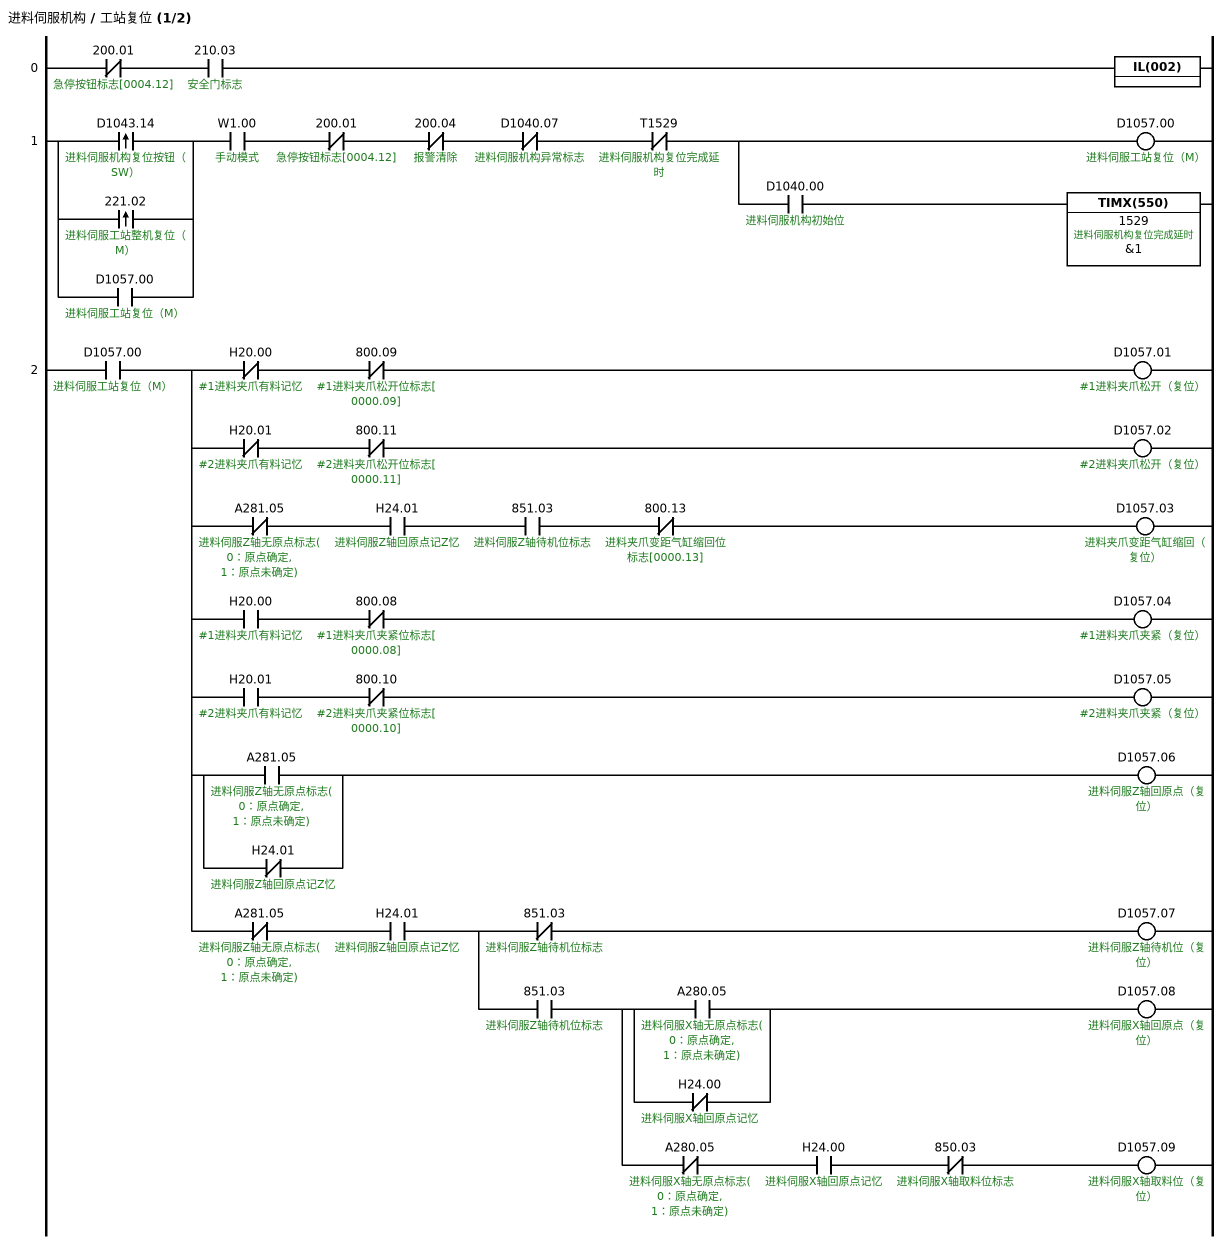
; rung 0
LDNOT 200.01  ; 急停按钮标志[0004.12]
AND 210.03  ; 安全门标志
IL(002)
; rung 1
@LD D1043.14  ; 进料伺服机构复位按钮（SW）
@OR 221.02  ; 进料伺服工站整机复位（M）
OR D1057.00  ; 进料伺服工站复位（M）
AND W1.00  ; 手动模式
ANDNOT 200.01  ; 急停按钮标志[0004.12]
ANDNOT 200.04  ; 报警清除
ANDNOT D1040.07  ; 进料伺服机构异常标志
ANDNOT T1529  ; 进料伺服机构复位完成延时
OUT D1057.00  ; 进料伺服工站复位（M）
AND D1040.00  ; 进料伺服机构初始位
TIMX(550) 1529 &1  ; 进料伺服机构复位完成延时
; rung 2
LD D1057.00  ; 进料伺服工站复位（M）
OUT TR0
ANDNOT H20.00  ; #1进料夹爪有料记忆
ANDNOT 800.09  ; #1进料夹爪松开位标志[0000.09]
OUT D1057.01  ; #1进料夹爪松开（复位）
LD TR0
ANDNOT H20.01  ; #2进料夹爪有料记忆
ANDNOT 800.11  ; #2进料夹爪松开位标志[0000.11]
OUT D1057.02  ; #2进料夹爪松开（复位）
LD TR0
ANDNOT A281.05  ; 进料伺服Z轴无原点标志(0：原点确定,1：原点未确定)
AND H24.01  ; 进料伺服Z轴回原点记Z忆
AND 851.03  ; 进料伺服Z轴待机位标志
ANDNOT 800.13  ; 进料夹爪变距气缸缩回位标志[0000.13]
OUT D1057.03  ; 进料夹爪变距气缸缩回（复位）
LD TR0
AND H20.00  ; #1进料夹爪有料记忆
ANDNOT 800.08  ; #1进料夹爪夹紧位标志[0000.08]
OUT D1057.04  ; #1进料夹爪夹紧（复位）
LD TR0
AND H20.01  ; #2进料夹爪有料记忆
ANDNOT 800.10  ; #2进料夹爪夹紧位标志[0000.10]
OUT D1057.05  ; #2进料夹爪夹紧（复位）
LD TR0
LD A281.05  ; 进料伺服Z轴无原点标志(0：原点确定,1：原点未确定)
ORNOT H24.01  ; 进料伺服Z轴回原点记Z忆
ANDLD
OUT D1057.06  ; 进料伺服Z轴回原点（复位）
LD TR0
ANDNOT A281.05  ; 进料伺服Z轴无原点标志(0：原点确定,1：原点未确定)
AND H24.01  ; 进料伺服Z轴回原点记Z忆
OUT TR0
ANDNOT 851.03  ; 进料伺服Z轴待机位标志
OUT D1057.07  ; 进料伺服Z轴待机位（复位）
LD TR0
AND 851.03  ; 进料伺服Z轴待机位标志
OUT TR0
LD A280.05  ; 进料伺服X轴无原点标志(0：原点确定,1：原点未确定)
ORNOT H24.00  ; 进料伺服X轴回原点记忆
ANDLD
OUT D1057.08  ; 进料伺服X轴回原点（复位）
LD TR0
ANDNOT A280.05  ; 进料伺服X轴无原点标志(0：原点确定,1：原点未确定)
AND H24.00  ; 进料伺服X轴回原点记忆
ANDNOT 850.03  ; 进料伺服X轴取料位标志
OUT D1057.09  ; 进料伺服X轴取料位（复位）

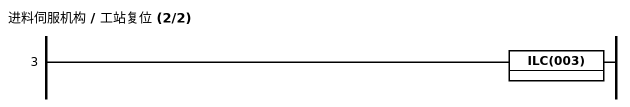
; rung 3
ILC(003)

### Section 指示灯

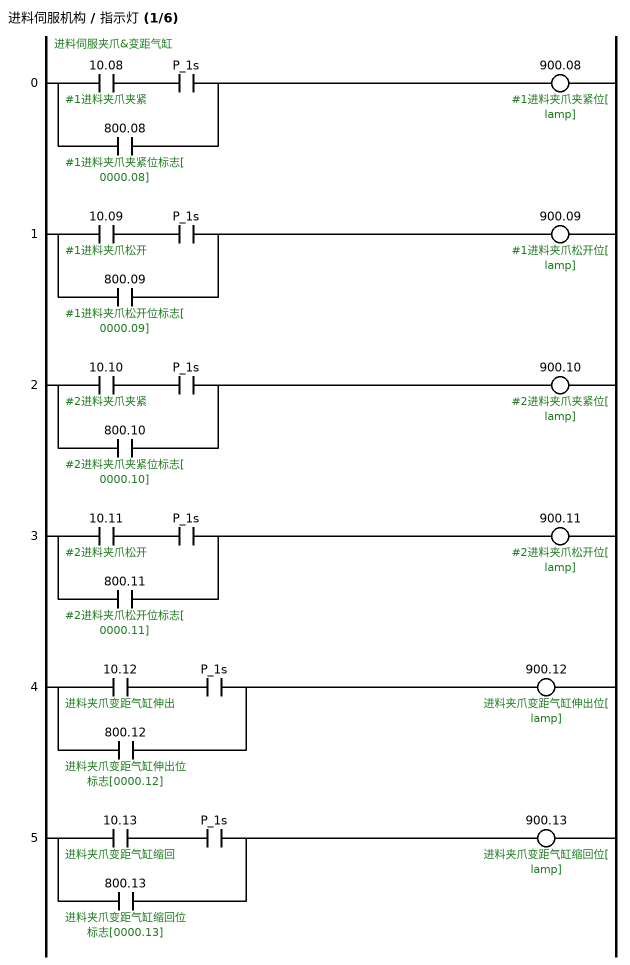
; rung 0: 进料伺服夹爪&变距气缸
LD 10.08  ; #1进料夹爪夹紧
AND P_1s
OR 800.08  ; #1进料夹爪夹紧位标志[0000.08]
OUT 900.08  ; #1进料夹爪夹紧位[lamp]
; rung 1
LD 10.09  ; #1进料夹爪松开
AND P_1s
OR 800.09  ; #1进料夹爪松开位标志[0000.09]
OUT 900.09  ; #1进料夹爪松开位[lamp]
; rung 2
LD 10.10  ; #2进料夹爪夹紧
AND P_1s
OR 800.10  ; #2进料夹爪夹紧位标志[0000.10]
OUT 900.10  ; #2进料夹爪夹紧位[lamp]
; rung 3
LD 10.11  ; #2进料夹爪松开
AND P_1s
OR 800.11  ; #2进料夹爪松开位标志[0000.11]
OUT 900.11  ; #2进料夹爪松开位[lamp]
; rung 4
LD 10.12  ; 进料夹爪变距气缸伸出
AND P_1s
OR 800.12  ; 进料夹爪变距气缸伸出位标志[0000.12]
OUT 900.12  ; 进料夹爪变距气缸伸出位[lamp]
; rung 5
LD 10.13  ; 进料夹爪变距气缸缩回
AND P_1s
OR 800.13  ; 进料夹爪变距气缸缩回位标志[0000.13]
OUT 900.13  ; 进料夹爪变距气缸缩回位[lamp]

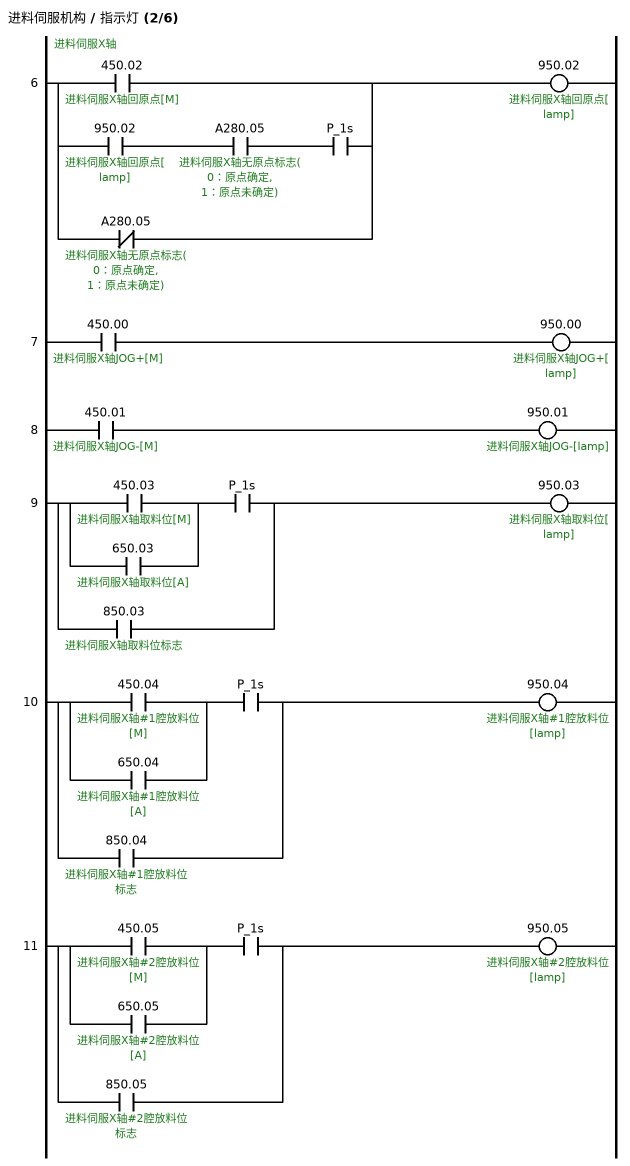
; rung 6: 进料伺服X轴
LD 450.02  ; 进料伺服X轴回原点[M]
LD 950.02  ; 进料伺服X轴回原点[lamp]
AND A280.05  ; 进料伺服X轴无原点标志(0：原点确定,1：原点未确定)
AND P_1s
ORLD
ORNOT A280.05  ; 进料伺服X轴无原点标志(0：原点确定,1：原点未确定)
OUT 950.02  ; 进料伺服X轴回原点[lamp]
; rung 7
LD 450.00  ; 进料伺服X轴JOG+[M]
OUT 950.00  ; 进料伺服X轴JOG+[lamp]
; rung 8
LD 450.01  ; 进料伺服X轴JOG-[M]
OUT 950.01  ; 进料伺服X轴JOG-[lamp]
; rung 9
LD 450.03  ; 进料伺服X轴取料位[M]
OR 650.03  ; 进料伺服X轴取料位[A]
AND P_1s
OR 850.03  ; 进料伺服X轴取料位标志
OUT 950.03  ; 进料伺服X轴取料位[lamp]
; rung 10
LD 450.04  ; 进料伺服X轴#1腔放料位[M]
OR 650.04  ; 进料伺服X轴#1腔放料位[A]
AND P_1s
OR 850.04  ; 进料伺服X轴#1腔放料位标志
OUT 950.04  ; 进料伺服X轴#1腔放料位[lamp]
; rung 11
LD 450.05  ; 进料伺服X轴#2腔放料位[M]
OR 650.05  ; 进料伺服X轴#2腔放料位[A]
AND P_1s
OR 850.05  ; 进料伺服X轴#2腔放料位标志
OUT 950.05  ; 进料伺服X轴#2腔放料位[lamp]

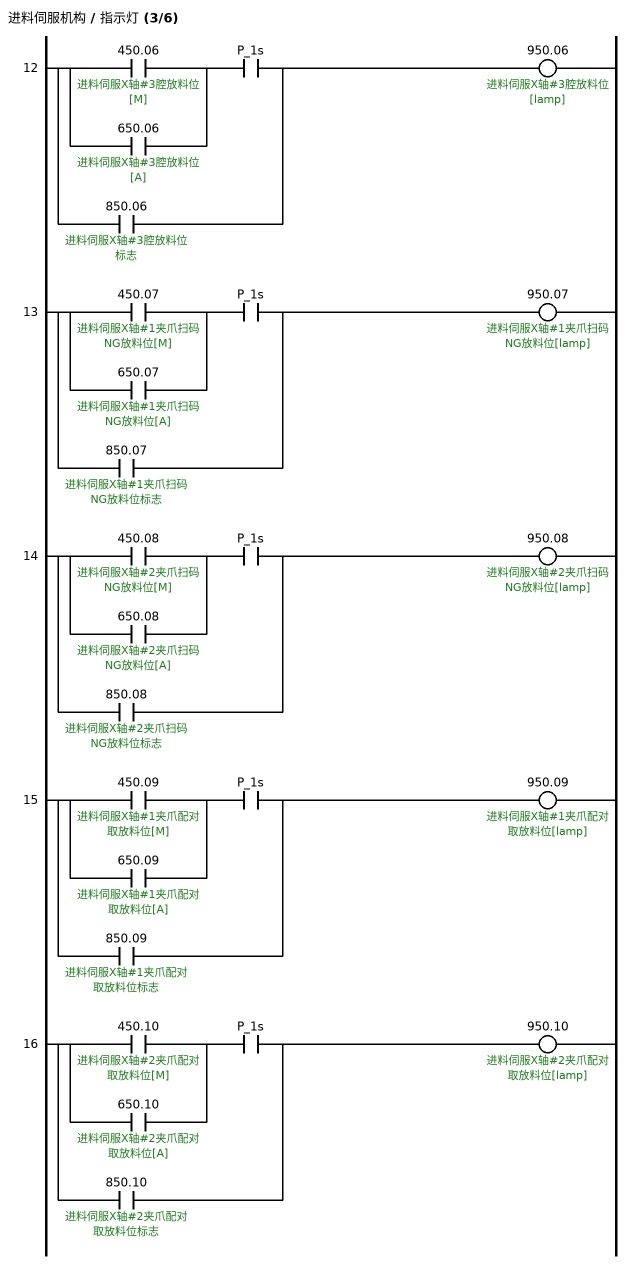
; rung 12
LD 450.06  ; 进料伺服X轴#3腔放料位[M]
OR 650.06  ; 进料伺服X轴#3腔放料位[A]
AND P_1s
OR 850.06  ; 进料伺服X轴#3腔放料位标志
OUT 950.06  ; 进料伺服X轴#3腔放料位[lamp]
; rung 13
LD 450.07  ; 进料伺服X轴#1夹爪扫码NG放料位[M]
OR 650.07  ; 进料伺服X轴#1夹爪扫码NG放料位[A]
AND P_1s
OR 850.07  ; 进料伺服X轴#1夹爪扫码NG放料位标志
OUT 950.07  ; 进料伺服X轴#1夹爪扫码NG放料位[lamp]
; rung 14
LD 450.08  ; 进料伺服X轴#2夹爪扫码NG放料位[M]
OR 650.08  ; 进料伺服X轴#2夹爪扫码NG放料位[A]
AND P_1s
OR 850.08  ; 进料伺服X轴#2夹爪扫码NG放料位标志
OUT 950.08  ; 进料伺服X轴#2夹爪扫码NG放料位[lamp]
; rung 15
LD 450.09  ; 进料伺服X轴#1夹爪配对取放料位[M]
OR 650.09  ; 进料伺服X轴#1夹爪配对取放料位[A]
AND P_1s
OR 850.09  ; 进料伺服X轴#1夹爪配对取放料位标志
OUT 950.09  ; 进料伺服X轴#1夹爪配对取放料位[lamp]
; rung 16
LD 450.10  ; 进料伺服X轴#2夹爪配对取放料位[M]
OR 650.10  ; 进料伺服X轴#2夹爪配对取放料位[A]
AND P_1s
OR 850.10  ; 进料伺服X轴#2夹爪配对取放料位标志
OUT 950.10  ; 进料伺服X轴#2夹爪配对取放料位[lamp]

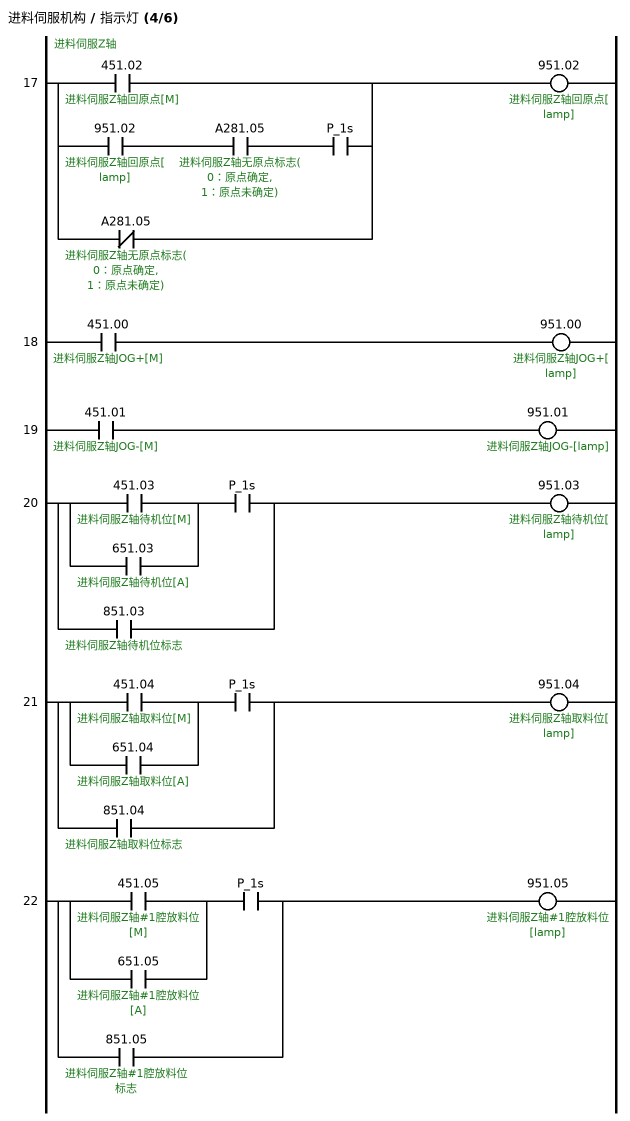
; rung 17: 进料伺服Z轴
LD 451.02  ; 进料伺服Z轴回原点[M]
LD 951.02  ; 进料伺服Z轴回原点[lamp]
AND A281.05  ; 进料伺服Z轴无原点标志(0：原点确定,1：原点未确定)
AND P_1s
ORLD
ORNOT A281.05  ; 进料伺服Z轴无原点标志(0：原点确定,1：原点未确定)
OUT 951.02  ; 进料伺服Z轴回原点[lamp]
; rung 18
LD 451.00  ; 进料伺服Z轴JOG+[M]
OUT 951.00  ; 进料伺服Z轴JOG+[lamp]
; rung 19
LD 451.01  ; 进料伺服Z轴JOG-[M]
OUT 951.01  ; 进料伺服Z轴JOG-[lamp]
; rung 20
LD 451.03  ; 进料伺服Z轴待机位[M]
OR 651.03  ; 进料伺服Z轴待机位[A]
AND P_1s
OR 851.03  ; 进料伺服Z轴待机位标志
OUT 951.03  ; 进料伺服Z轴待机位[lamp]
; rung 21
LD 451.04  ; 进料伺服Z轴取料位[M]
OR 651.04  ; 进料伺服Z轴取料位[A]
AND P_1s
OR 851.04  ; 进料伺服Z轴取料位标志
OUT 951.04  ; 进料伺服Z轴取料位[lamp]
; rung 22
LD 451.05  ; 进料伺服Z轴#1腔放料位[M]
OR 651.05  ; 进料伺服Z轴#1腔放料位[A]
AND P_1s
OR 851.05  ; 进料伺服Z轴#1腔放料位标志
OUT 951.05  ; 进料伺服Z轴#1腔放料位[lamp]

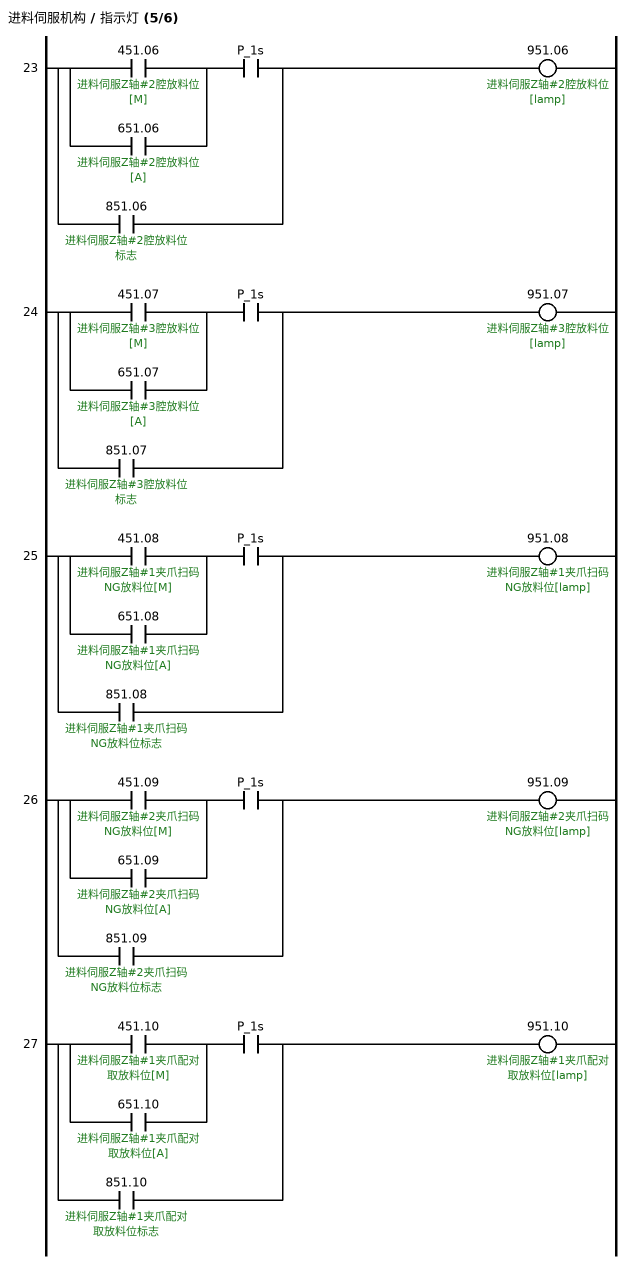
; rung 23
LD 451.06  ; 进料伺服Z轴#2腔放料位[M]
OR 651.06  ; 进料伺服Z轴#2腔放料位[A]
AND P_1s
OR 851.06  ; 进料伺服Z轴#2腔放料位标志
OUT 951.06  ; 进料伺服Z轴#2腔放料位[lamp]
; rung 24
LD 451.07  ; 进料伺服Z轴#3腔放料位[M]
OR 651.07  ; 进料伺服Z轴#3腔放料位[A]
AND P_1s
OR 851.07  ; 进料伺服Z轴#3腔放料位标志
OUT 951.07  ; 进料伺服Z轴#3腔放料位[lamp]
; rung 25
LD 451.08  ; 进料伺服Z轴#1夹爪扫码NG放料位[M]
OR 651.08  ; 进料伺服Z轴#1夹爪扫码NG放料位[A]
AND P_1s
OR 851.08  ; 进料伺服Z轴#1夹爪扫码NG放料位标志
OUT 951.08  ; 进料伺服Z轴#1夹爪扫码NG放料位[lamp]
; rung 26
LD 451.09  ; 进料伺服Z轴#2夹爪扫码NG放料位[M]
OR 651.09  ; 进料伺服Z轴#2夹爪扫码NG放料位[A]
AND P_1s
OR 851.09  ; 进料伺服Z轴#2夹爪扫码NG放料位标志
OUT 951.09  ; 进料伺服Z轴#2夹爪扫码NG放料位[lamp]
; rung 27
LD 451.10  ; 进料伺服Z轴#1夹爪配对取放料位[M]
OR 651.10  ; 进料伺服Z轴#1夹爪配对取放料位[A]
AND P_1s
OR 851.10  ; 进料伺服Z轴#1夹爪配对取放料位标志
OUT 951.10  ; 进料伺服Z轴#1夹爪配对取放料位[lamp]

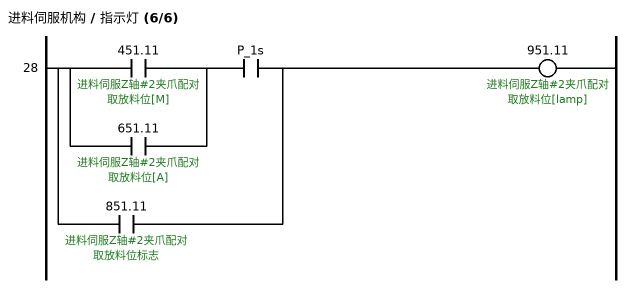
; rung 28
LD 451.11  ; 进料伺服Z轴#2夹爪配对取放料位[M]
OR 651.11  ; 进料伺服Z轴#2夹爪配对取放料位[A]
AND P_1s
OR 851.11  ; 进料伺服Z轴#2夹爪配对取放料位标志
OUT 951.11  ; 进料伺服Z轴#2夹爪配对取放料位[lamp]

### Section 外部输出

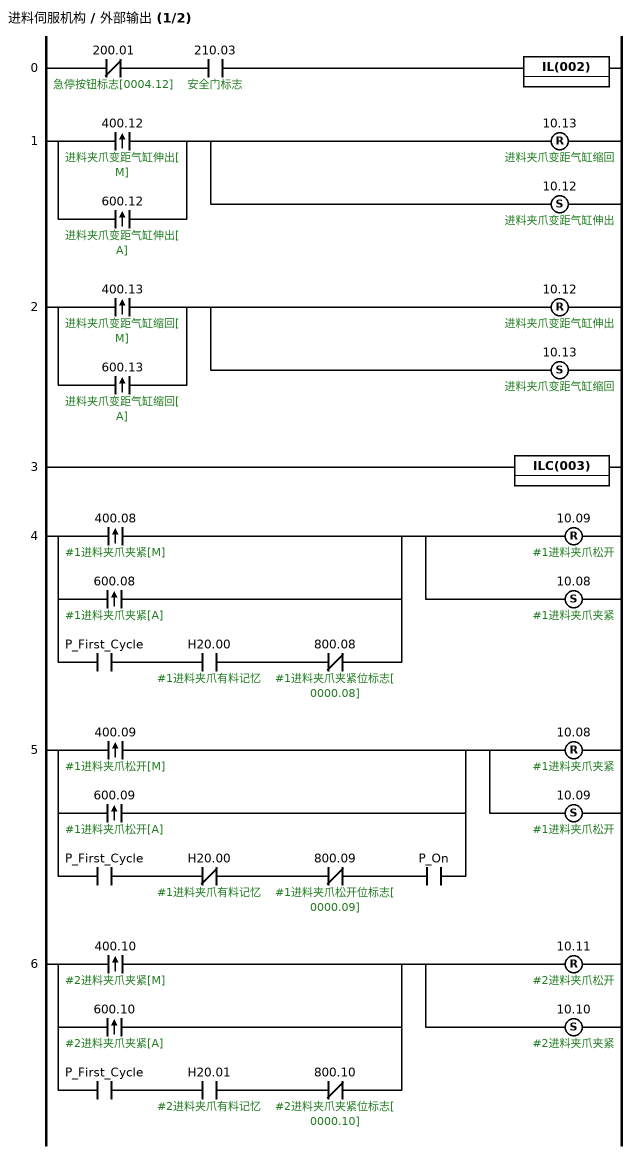
; rung 0
LDNOT 200.01  ; 急停按钮标志[0004.12]
AND 210.03  ; 安全门标志
IL(002)
; rung 1
@LD 400.12  ; 进料夹爪变距气缸伸出[M]
@OR 600.12  ; 进料夹爪变距气缸伸出[A]
RSET 10.13  ; 进料夹爪变距气缸缩回
SET 10.12  ; 进料夹爪变距气缸伸出
; rung 2
@LD 400.13  ; 进料夹爪变距气缸缩回[M]
@OR 600.13  ; 进料夹爪变距气缸缩回[A]
RSET 10.12  ; 进料夹爪变距气缸伸出
SET 10.13  ; 进料夹爪变距气缸缩回
; rung 3
ILC(003)
; rung 4
@LD 400.08  ; #1进料夹爪夹紧[M]
@OR 600.08  ; #1进料夹爪夹紧[A]
LD P_First_Cycle
AND H20.00  ; #1进料夹爪有料记忆
ANDNOT 800.08  ; #1进料夹爪夹紧位标志[0000.08]
ORLD
RSET 10.09  ; #1进料夹爪松开
SET 10.08  ; #1进料夹爪夹紧
; rung 5
@LD 400.09  ; #1进料夹爪松开[M]
@OR 600.09  ; #1进料夹爪松开[A]
LD P_First_Cycle
ANDNOT H20.00  ; #1进料夹爪有料记忆
ANDNOT 800.09  ; #1进料夹爪松开位标志[0000.09]
AND P_On
ORLD
RSET 10.08  ; #1进料夹爪夹紧
SET 10.09  ; #1进料夹爪松开
; rung 6
@LD 400.10  ; #2进料夹爪夹紧[M]
@OR 600.10  ; #2进料夹爪夹紧[A]
LD P_First_Cycle
AND H20.01  ; #2进料夹爪有料记忆
ANDNOT 800.10  ; #2进料夹爪夹紧位标志[0000.10]
ORLD
RSET 10.11  ; #2进料夹爪松开
SET 10.10  ; #2进料夹爪夹紧

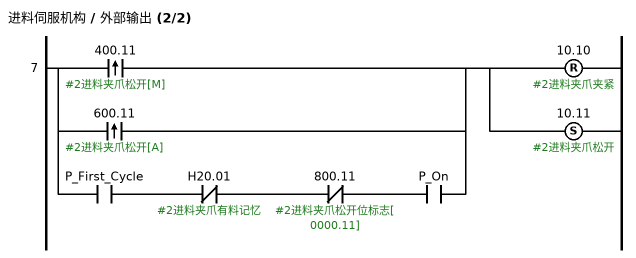
; rung 7
@LD 400.11  ; #2进料夹爪松开[M]
@OR 600.11  ; #2进料夹爪松开[A]
LD P_First_Cycle
ANDNOT H20.01  ; #2进料夹爪有料记忆
ANDNOT 800.11  ; #2进料夹爪松开位标志[0000.11]
AND P_On
ORLD
RSET 10.10  ; #2进料夹爪夹紧
SET 10.11  ; #2进料夹爪松开

### Section END
; rung 0
END(001)

## Program 氦检机构 (cyclic task 3)
Local symbols
UP BOOL

### Section Main

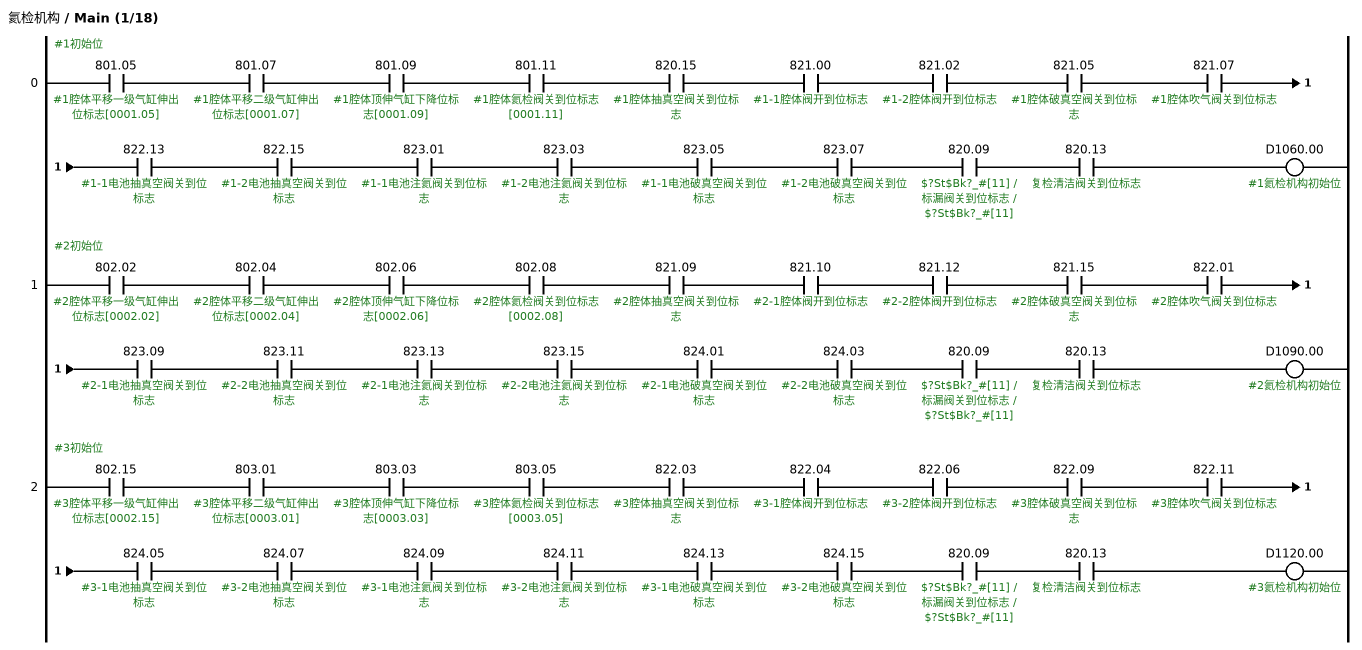
; rung 0: #1初始位
LD 801.05  ; #1腔体平移一级气缸伸出位标志[0001.05]
AND 801.07  ; #1腔体平移二级气缸伸出位标志[0001.07]
AND 801.09  ; #1腔体顶伸气缸下降位标志[0001.09]
AND 801.11  ; #1腔体氦检阀关到位标志[0001.11]
AND 820.15  ; #1腔体抽真空阀关到位标志
AND 821.00  ; #1-1腔体阀开到位标志
AND 821.02  ; #1-2腔体阀开到位标志
AND 821.05  ; #1腔体破真空阀关到位标志
AND 821.07  ; #1腔体吹气阀关到位标志
AND 822.13  ; #1-1电池抽真空阀关到位标志
AND 822.15  ; #1-2电池抽真空阀关到位标志
AND 823.01  ; #1-1电池注氦阀关到位标志
AND 823.03  ; #1-2电池注氦阀关到位标志
AND 823.05  ; #1-1电池破真空阀关到位标志
AND 823.07  ; #1-2电池破真空阀关到位标志
AND 820.09  ; $?St$Bk?_#[11] / 标漏阀关到位标志 / $?St$Bk?_#[11]
AND 820.13  ; 复检清洁阀关到位标志
OUT D1060.00  ; #1氦检机构初始位
; rung 1: #2初始位
LD 802.02  ; #2腔体平移一级气缸伸出位标志[0002.02]
AND 802.04  ; #2腔体平移二级气缸伸出位标志[0002.04]
AND 802.06  ; #2腔体顶伸气缸下降位标志[0002.06]
AND 802.08  ; #2腔体氦检阀关到位标志[0002.08]
AND 821.09  ; #2腔体抽真空阀关到位标志
AND 821.10  ; #2-1腔体阀开到位标志
AND 821.12  ; #2-2腔体阀开到位标志
AND 821.15  ; #2腔体破真空阀关到位标志
AND 822.01  ; #2腔体吹气阀关到位标志
AND 823.09  ; #2-1电池抽真空阀关到位标志
AND 823.11  ; #2-2电池抽真空阀关到位标志
AND 823.13  ; #2-1电池注氦阀关到位标志
AND 823.15  ; #2-2电池注氦阀关到位标志
AND 824.01  ; #2-1电池破真空阀关到位标志
AND 824.03  ; #2-2电池破真空阀关到位标志
AND 820.09  ; $?St$Bk?_#[11] / 标漏阀关到位标志 / $?St$Bk?_#[11]
AND 820.13  ; 复检清洁阀关到位标志
OUT D1090.00  ; #2氦检机构初始位
; rung 2: #3初始位
LD 802.15  ; #3腔体平移一级气缸伸出位标志[0002.15]
AND 803.01  ; #3腔体平移二级气缸伸出位标志[0003.01]
AND 803.03  ; #3腔体顶伸气缸下降位标志[0003.03]
AND 803.05  ; #3腔体氦检阀关到位标志[0003.05]
AND 822.03  ; #3腔体抽真空阀关到位标志
AND 822.04  ; #3-1腔体阀开到位标志
AND 822.06  ; #3-2腔体阀开到位标志
AND 822.09  ; #3腔体破真空阀关到位标志
AND 822.11  ; #3腔体吹气阀关到位标志
AND 824.05  ; #3-1电池抽真空阀关到位标志
AND 824.07  ; #3-2电池抽真空阀关到位标志
AND 824.09  ; #3-1电池注氦阀关到位标志
AND 824.11  ; #3-2电池注氦阀关到位标志
AND 824.13  ; #3-1电池破真空阀关到位标志
AND 824.15  ; #3-2电池破真空阀关到位标志
AND 820.09  ; $?St$Bk?_#[11] / 标漏阀关到位标志 / $?St$Bk?_#[11]
AND 820.13  ; 复检清洁阀关到位标志
OUT D1120.00  ; #3氦检机构初始位

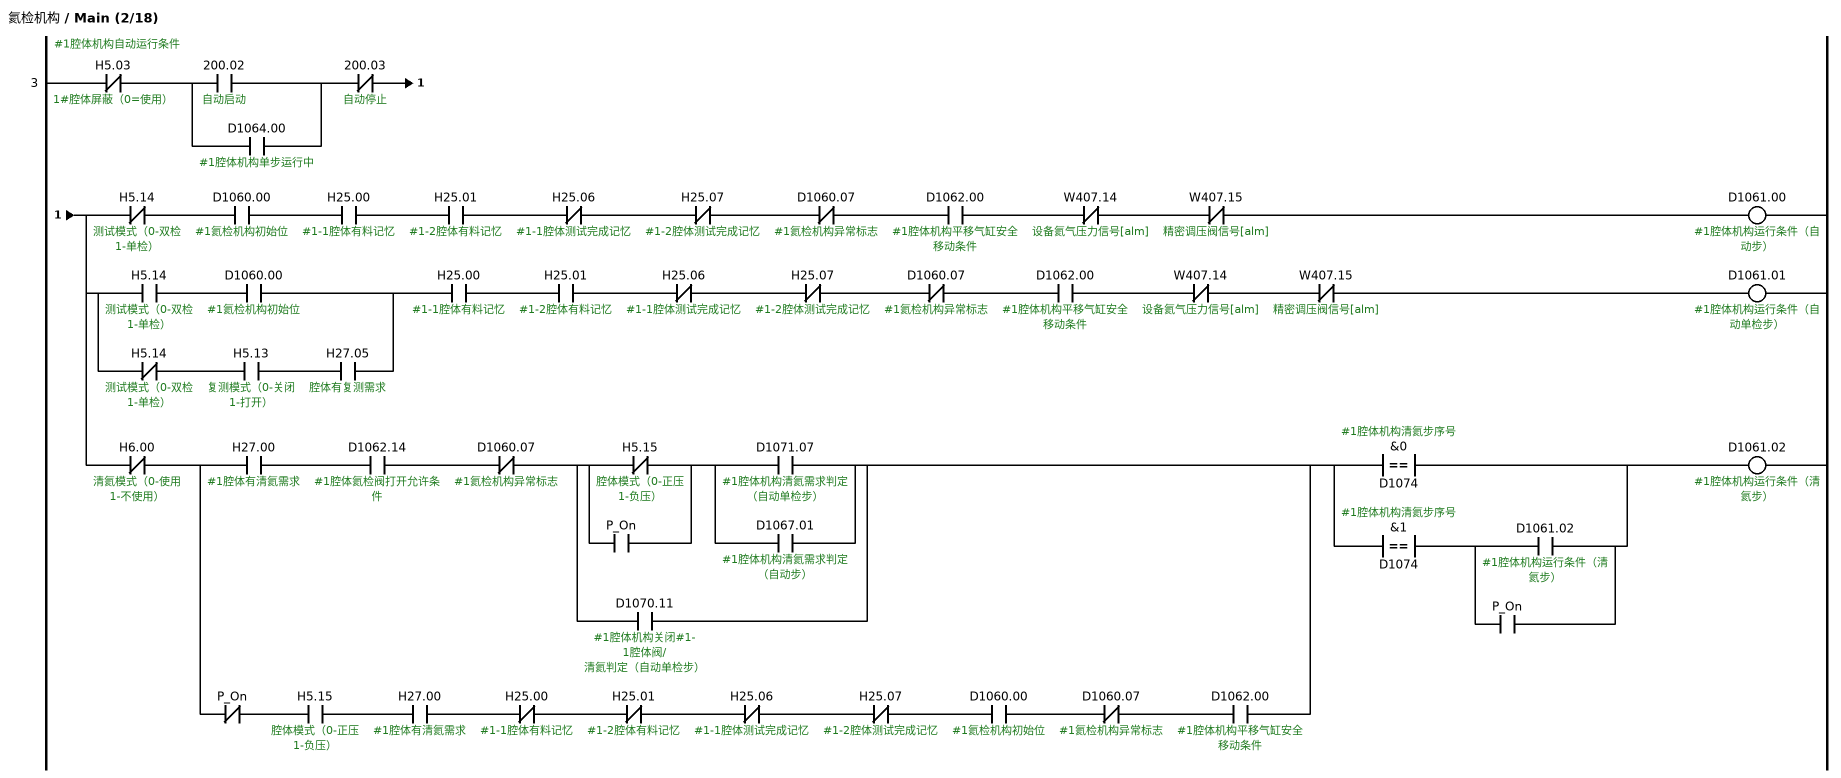
; rung 3: #1腔体机构自动运行条件
LDNOT H5.03  ; 1#腔体屏蔽（0=使用）
LD 200.02  ; 自动启动
OR D1064.00  ; #1腔体机构单步运行中
ANDLD
ANDNOT 200.03  ; 自动停止
OUT TR0
ANDNOT H5.14  ; 测试模式（0-双检 1-单检）
AND D1060.00  ; #1氦检机构初始位
AND H25.00  ; #1-1腔体有料记忆
AND H25.01  ; #1-2腔体有料记忆
ANDNOT H25.06  ; #1-1腔体测试完成记忆
ANDNOT H25.07  ; #1-2腔体测试完成记忆
ANDNOT D1060.07  ; #1氦检机构异常标志
AND D1062.00  ; #1腔体机构平移气缸安全移动条件
ANDNOT W407.14  ; 设备氦气压力信号[alm]
ANDNOT W407.15  ; 精密调压阀信号[alm]
OUT D1061.00  ; #1腔体机构运行条件（自动步）
LD TR0
LD H5.14  ; 测试模式（0-双检 1-单检）
AND D1060.00  ; #1氦检机构初始位
LDNOT H5.14  ; 测试模式（0-双检 1-单检）
AND H5.13  ; 复测模式（0-关闭 1-打开）
AND H27.05  ; 腔体有复测需求
ORLD
ANDLD
AND H25.00  ; #1-1腔体有料记忆
AND H25.01  ; #1-2腔体有料记忆
ANDNOT H25.06  ; #1-1腔体测试完成记忆
ANDNOT H25.07  ; #1-2腔体测试完成记忆
ANDNOT D1060.07  ; #1氦检机构异常标志
AND D1062.00  ; #1腔体机构平移气缸安全移动条件
ANDNOT W407.14  ; 设备氦气压力信号[alm]
ANDNOT W407.15  ; 精密调压阀信号[alm]
OUT D1061.01  ; #1腔体机构运行条件（自动单检步）
LD TR0
ANDNOT H6.00  ; 清氦模式（0-使用 1-不使用）
LD H27.00  ; #1腔体有清氦需求
AND D1062.14  ; #1腔体氦检阀打开允许条件
ANDNOT D1060.07  ; #1氦检机构异常标志
LDNOT H5.15  ; 腔体模式（0-正压 1-负压）
OR P_On
LD D1071.07  ; #1腔体机构清氦需求判定（自动单检步）
OR D1067.01  ; #1腔体机构清氦需求判定（自动步）
ANDLD
OR D1070.11  ; #1腔体机构关闭#1-1腔体阀/清氦判定（自动单检步）
ANDLD
LDNOT P_On
AND H5.15  ; 腔体模式（0-正压 1-负压）
AND H27.00  ; #1腔体有清氦需求
ANDNOT H25.00  ; #1-1腔体有料记忆
ANDNOT H25.01  ; #1-2腔体有料记忆
ANDNOT H25.06  ; #1-1腔体测试完成记忆
ANDNOT H25.07  ; #1-2腔体测试完成记忆
AND D1060.00  ; #1氦检机构初始位
ANDNOT D1060.07  ; #1氦检机构异常标志
AND D1062.00  ; #1腔体机构平移气缸安全移动条件
ORLD
ANDLD
LD=L(301) &0 D1074  ; #1腔体机构清氦步序号
LD=L(301) &1 D1074  ; #1腔体机构清氦步序号
LD D1061.02  ; #1腔体机构运行条件（清氦步）
OR P_On
ANDLD
ORLD
ANDLD
OUT D1061.02  ; #1腔体机构运行条件（清氦步）

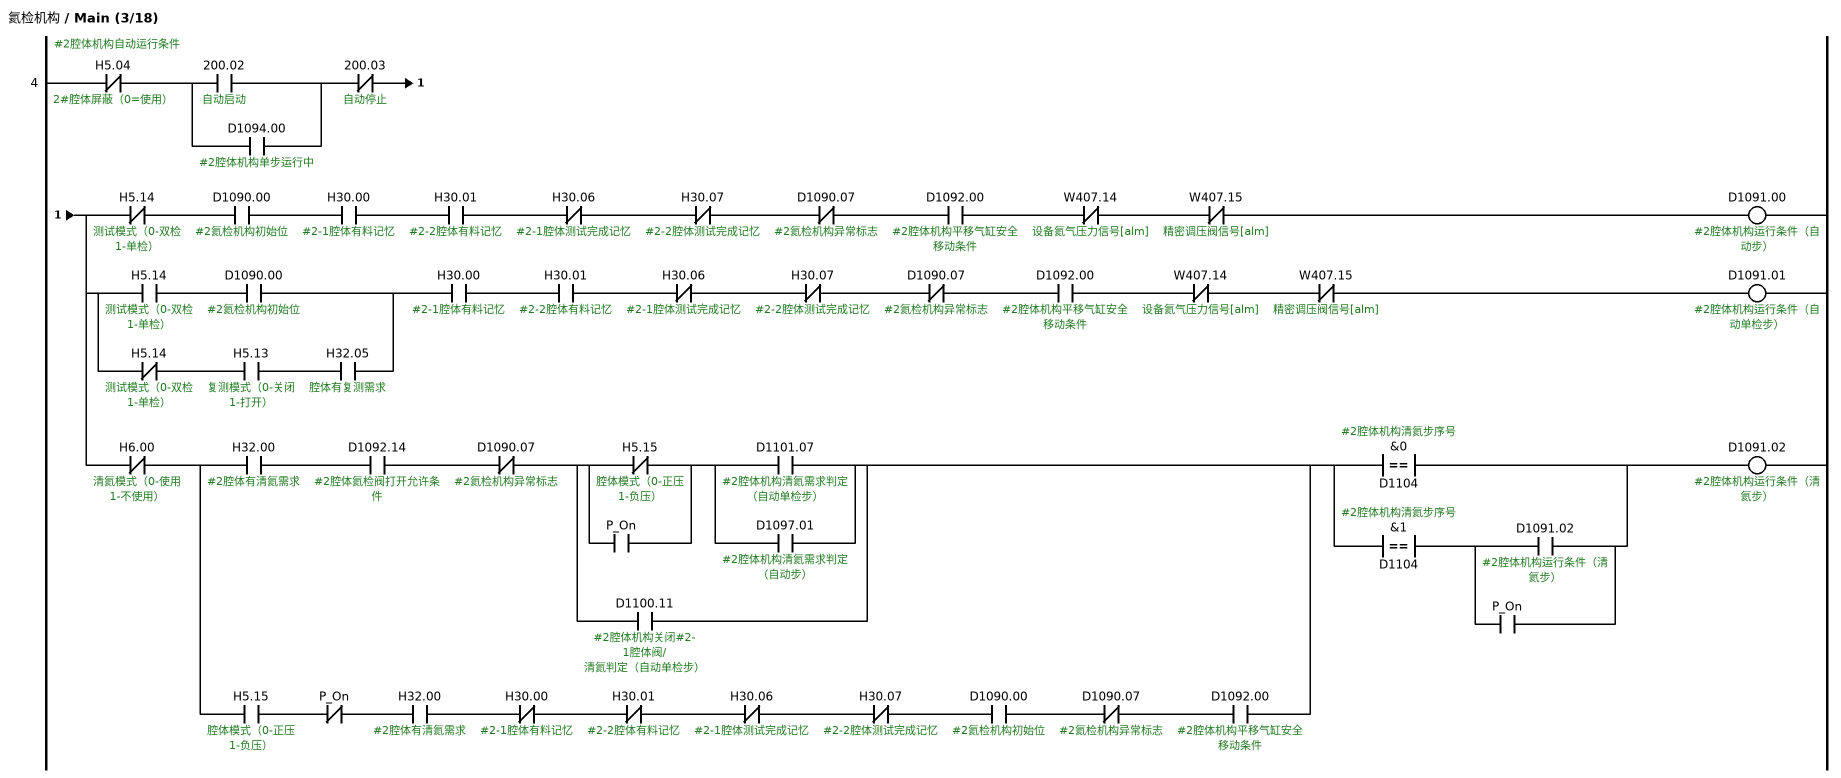
; rung 4: #2腔体机构自动运行条件
LDNOT H5.04  ; 2#腔体屏蔽（0=使用）
LD 200.02  ; 自动启动
OR D1094.00  ; #2腔体机构单步运行中
ANDLD
ANDNOT 200.03  ; 自动停止
OUT TR0
ANDNOT H5.14  ; 测试模式（0-双检 1-单检）
AND D1090.00  ; #2氦检机构初始位
AND H30.00  ; #2-1腔体有料记忆
AND H30.01  ; #2-2腔体有料记忆
ANDNOT H30.06  ; #2-1腔体测试完成记忆
ANDNOT H30.07  ; #2-2腔体测试完成记忆
ANDNOT D1090.07  ; #2氦检机构异常标志
AND D1092.00  ; #2腔体机构平移气缸安全移动条件
ANDNOT W407.14  ; 设备氦气压力信号[alm]
ANDNOT W407.15  ; 精密调压阀信号[alm]
OUT D1091.00  ; #2腔体机构运行条件（自动步）
LD TR0
LD H5.14  ; 测试模式（0-双检 1-单检）
AND D1090.00  ; #2氦检机构初始位
LDNOT H5.14  ; 测试模式（0-双检 1-单检）
AND H5.13  ; 复测模式（0-关闭 1-打开）
AND H32.05  ; 腔体有复测需求
ORLD
ANDLD
AND H30.00  ; #2-1腔体有料记忆
AND H30.01  ; #2-2腔体有料记忆
ANDNOT H30.06  ; #2-1腔体测试完成记忆
ANDNOT H30.07  ; #2-2腔体测试完成记忆
ANDNOT D1090.07  ; #2氦检机构异常标志
AND D1092.00  ; #2腔体机构平移气缸安全移动条件
ANDNOT W407.14  ; 设备氦气压力信号[alm]
ANDNOT W407.15  ; 精密调压阀信号[alm]
OUT D1091.01  ; #2腔体机构运行条件（自动单检步）
LD TR0
ANDNOT H6.00  ; 清氦模式（0-使用 1-不使用）
LD H32.00  ; #2腔体有清氦需求
AND D1092.14  ; #2腔体氦检阀打开允许条件
ANDNOT D1090.07  ; #2氦检机构异常标志
LDNOT H5.15  ; 腔体模式（0-正压 1-负压）
OR P_On
LD D1101.07  ; #2腔体机构清氦需求判定（自动单检步）
OR D1097.01  ; #2腔体机构清氦需求判定（自动步）
ANDLD
OR D1100.11  ; #2腔体机构关闭#2-1腔体阀/清氦判定（自动单检步）
ANDLD
LD H5.15  ; 腔体模式（0-正压 1-负压）
ANDNOT P_On
AND H32.00  ; #2腔体有清氦需求
ANDNOT H30.00  ; #2-1腔体有料记忆
ANDNOT H30.01  ; #2-2腔体有料记忆
ANDNOT H30.06  ; #2-1腔体测试完成记忆
ANDNOT H30.07  ; #2-2腔体测试完成记忆
AND D1090.00  ; #2氦检机构初始位
ANDNOT D1090.07  ; #2氦检机构异常标志
AND D1092.00  ; #2腔体机构平移气缸安全移动条件
ORLD
ANDLD
LD=L(301) &0 D1104  ; #2腔体机构清氦步序号
LD=L(301) &1 D1104  ; #2腔体机构清氦步序号
LD D1091.02  ; #2腔体机构运行条件（清氦步）
OR P_On
ANDLD
ORLD
ANDLD
OUT D1091.02  ; #2腔体机构运行条件（清氦步）

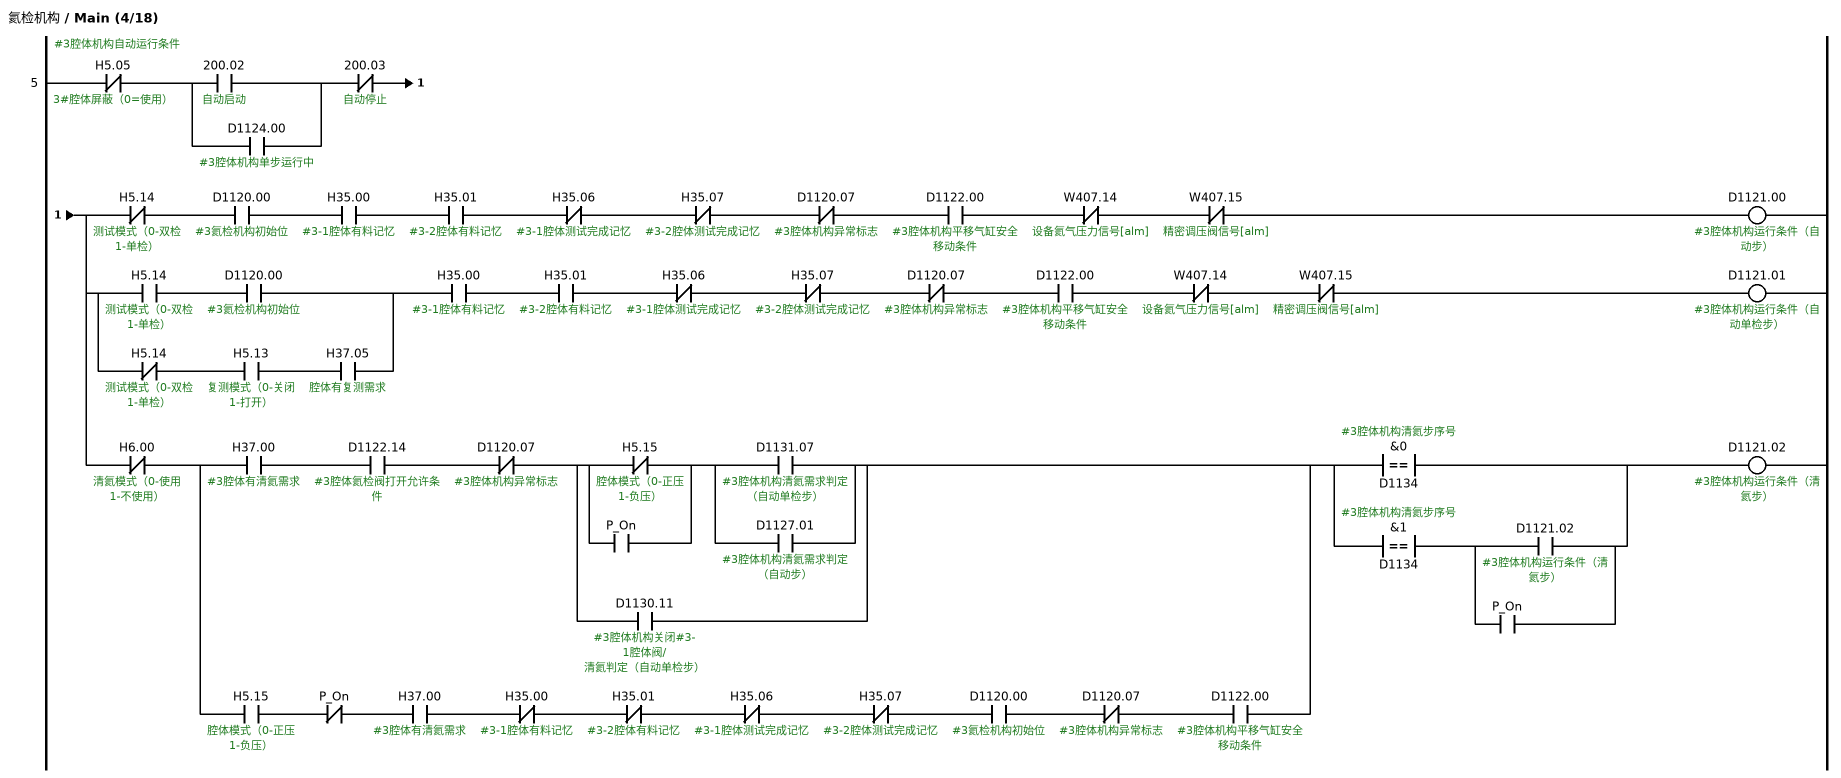
; rung 5: #3腔体机构自动运行条件
LDNOT H5.05  ; 3#腔体屏蔽（0=使用）
LD 200.02  ; 自动启动
OR D1124.00  ; #3腔体机构单步运行中
ANDLD
ANDNOT 200.03  ; 自动停止
OUT TR0
ANDNOT H5.14  ; 测试模式（0-双检 1-单检）
AND D1120.00  ; #3氦检机构初始位
AND H35.00  ; #3-1腔体有料记忆
AND H35.01  ; #3-2腔体有料记忆
ANDNOT H35.06  ; #3-1腔体测试完成记忆
ANDNOT H35.07  ; #3-2腔体测试完成记忆
ANDNOT D1120.07  ; #3腔体机构异常标志
AND D1122.00  ; #3腔体机构平移气缸安全移动条件
ANDNOT W407.14  ; 设备氦气压力信号[alm]
ANDNOT W407.15  ; 精密调压阀信号[alm]
OUT D1121.00  ; #3腔体机构运行条件（自动步）
LD TR0
LD H5.14  ; 测试模式（0-双检 1-单检）
AND D1120.00  ; #3氦检机构初始位
LDNOT H5.14  ; 测试模式（0-双检 1-单检）
AND H5.13  ; 复测模式（0-关闭 1-打开）
AND H37.05  ; 腔体有复测需求
ORLD
ANDLD
AND H35.00  ; #3-1腔体有料记忆
AND H35.01  ; #3-2腔体有料记忆
ANDNOT H35.06  ; #3-1腔体测试完成记忆
ANDNOT H35.07  ; #3-2腔体测试完成记忆
ANDNOT D1120.07  ; #3腔体机构异常标志
AND D1122.00  ; #3腔体机构平移气缸安全移动条件
ANDNOT W407.14  ; 设备氦气压力信号[alm]
ANDNOT W407.15  ; 精密调压阀信号[alm]
OUT D1121.01  ; #3腔体机构运行条件（自动单检步）
LD TR0
ANDNOT H6.00  ; 清氦模式（0-使用 1-不使用）
LD H37.00  ; #3腔体有清氦需求
AND D1122.14  ; #3腔体氦检阀打开允许条件
ANDNOT D1120.07  ; #3腔体机构异常标志
LDNOT H5.15  ; 腔体模式（0-正压 1-负压）
OR P_On
LD D1131.07  ; #3腔体机构清氦需求判定（自动单检步）
OR D1127.01  ; #3腔体机构清氦需求判定（自动步）
ANDLD
OR D1130.11  ; #3腔体机构关闭#3-1腔体阀/清氦判定（自动单检步）
ANDLD
LD H5.15  ; 腔体模式（0-正压 1-负压）
ANDNOT P_On
AND H37.00  ; #3腔体有清氦需求
ANDNOT H35.00  ; #3-1腔体有料记忆
ANDNOT H35.01  ; #3-2腔体有料记忆
ANDNOT H35.06  ; #3-1腔体测试完成记忆
ANDNOT H35.07  ; #3-2腔体测试完成记忆
AND D1120.00  ; #3氦检机构初始位
ANDNOT D1120.07  ; #3腔体机构异常标志
AND D1122.00  ; #3腔体机构平移气缸安全移动条件
ORLD
ANDLD
LD=L(301) &0 D1134  ; #3腔体机构清氦步序号
LD=L(301) &1 D1134  ; #3腔体机构清氦步序号
LD D1121.02  ; #3腔体机构运行条件（清氦步）
OR P_On
ANDLD
ORLD
ANDLD
OUT D1121.02  ; #3腔体机构运行条件（清氦步）

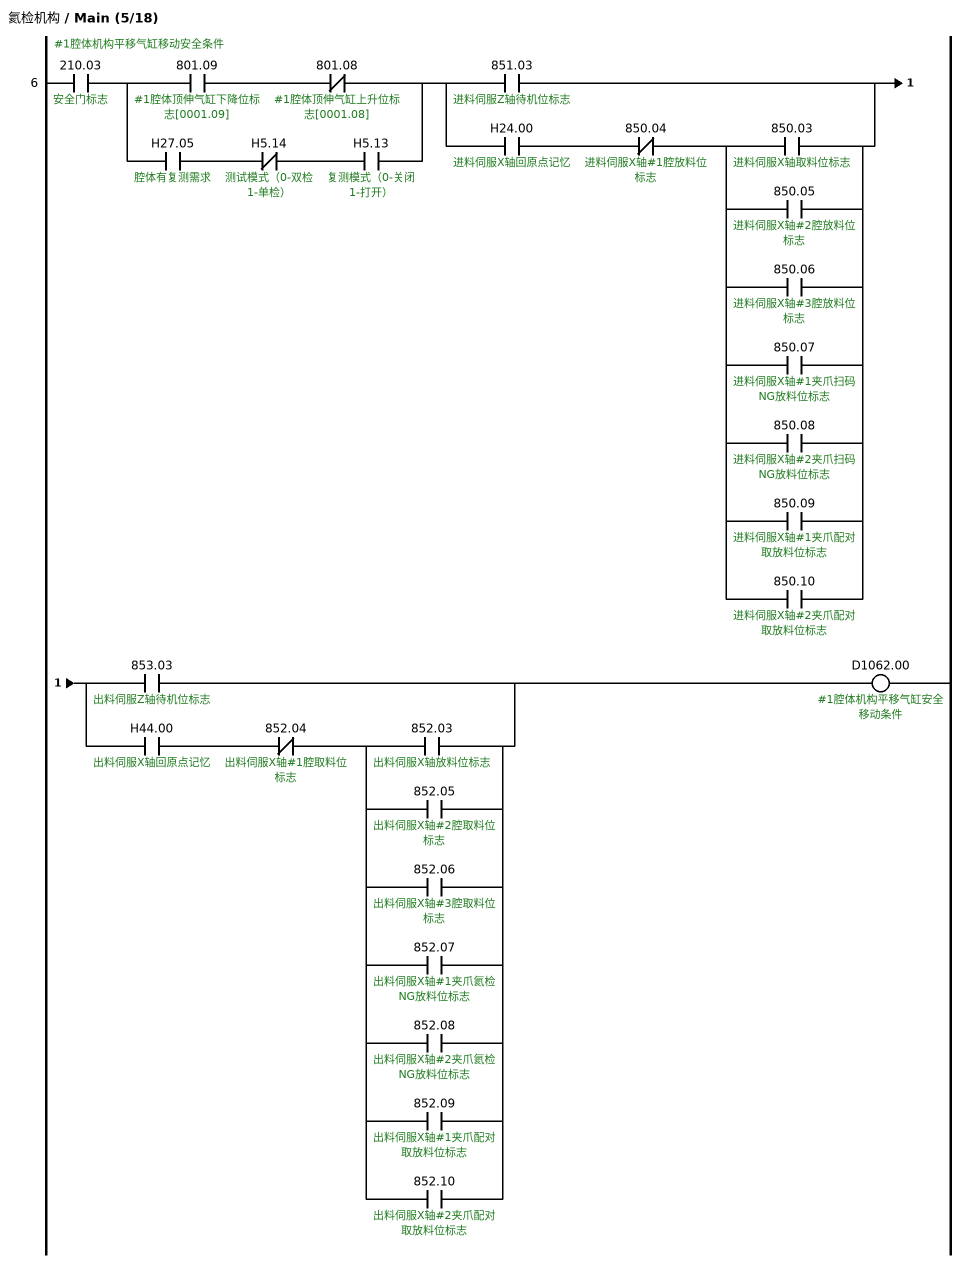
; rung 6: #1腔体机构平移气缸移动安全条件
LD 210.03  ; 安全门标志
LD 801.09  ; #1腔体顶伸气缸下降位标志[0001.09]
ANDNOT 801.08  ; #1腔体顶伸气缸上升位标志[0001.08]
LD H27.05  ; 腔体有复测需求
ANDNOT H5.14  ; 测试模式（0-双检 1-单检）
AND H5.13  ; 复测模式（0-关闭 1-打开）
ORLD
ANDLD
LD 851.03  ; 进料伺服Z轴待机位标志
LD H24.00  ; 进料伺服X轴回原点记忆
ANDNOT 850.04  ; 进料伺服X轴#1腔放料位标志
LD 850.03  ; 进料伺服X轴取料位标志
OR 850.05  ; 进料伺服X轴#2腔放料位标志
OR 850.06  ; 进料伺服X轴#3腔放料位标志
OR 850.07  ; 进料伺服X轴#1夹爪扫码NG放料位标志
OR 850.08  ; 进料伺服X轴#2夹爪扫码NG放料位标志
OR 850.09  ; 进料伺服X轴#1夹爪配对取放料位标志
OR 850.10  ; 进料伺服X轴#2夹爪配对取放料位标志
ANDLD
ORLD
ANDLD
LD 853.03  ; 出料伺服Z轴待机位标志
LD H44.00  ; 出料伺服X轴回原点记忆
ANDNOT 852.04  ; 出料伺服X轴#1腔取料位标志
LD 852.03  ; 出料伺服X轴放料位标志
OR 852.05  ; 出料伺服X轴#2腔取料位标志
OR 852.06  ; 出料伺服X轴#3腔取料位标志
OR 852.07  ; 出料伺服X轴#1夹爪氦检NG放料位标志
OR 852.08  ; 出料伺服X轴#2夹爪氦检NG放料位标志
OR 852.09  ; 出料伺服X轴#1夹爪配对取放料位标志
OR 852.10  ; 出料伺服X轴#2夹爪配对取放料位标志
ANDLD
ORLD
ANDLD
OUT D1062.00  ; #1腔体机构平移气缸安全移动条件

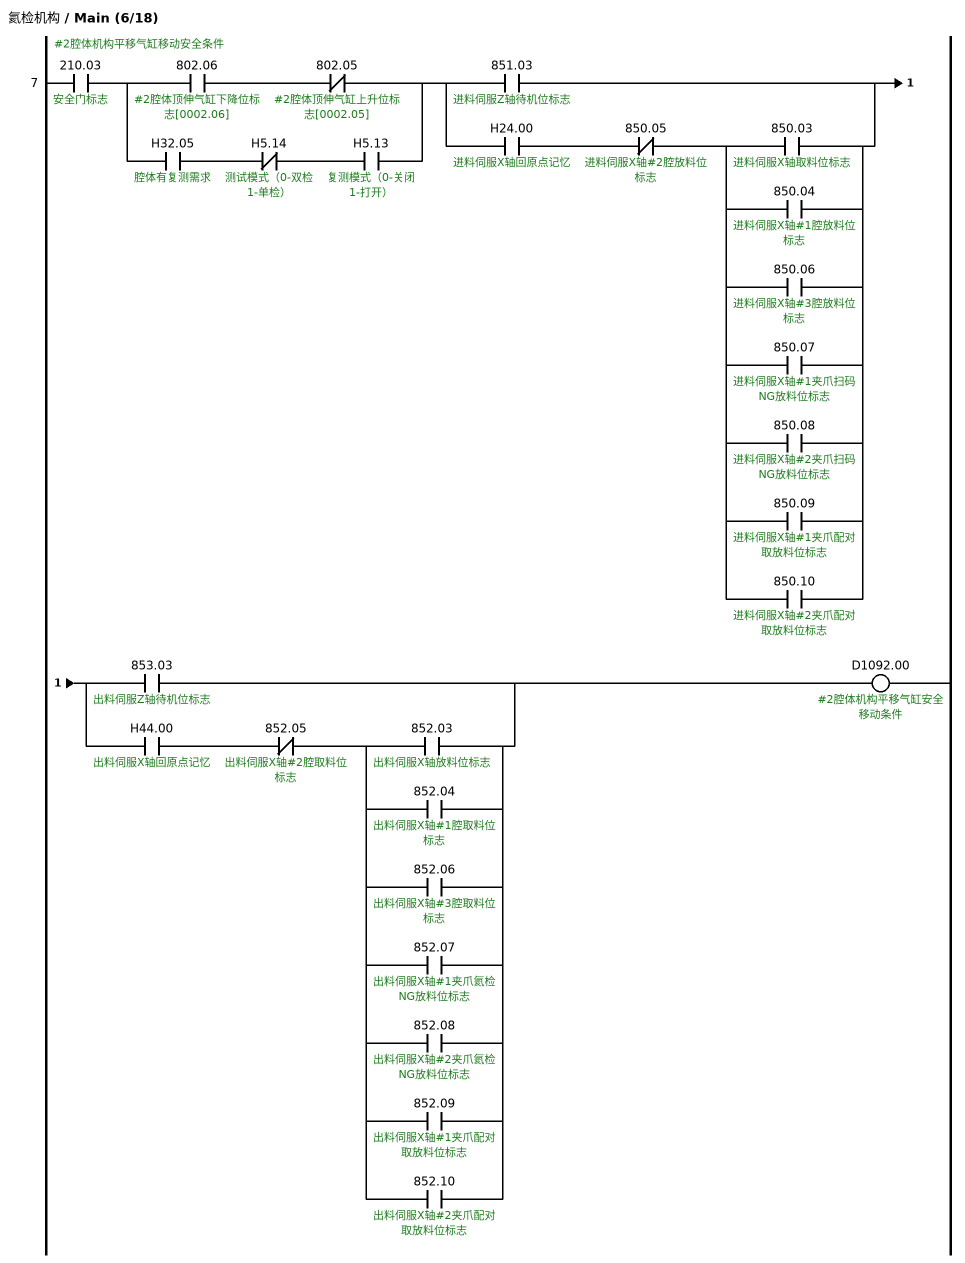
; rung 7: #2腔体机构平移气缸移动安全条件
LD 210.03  ; 安全门标志
LD 802.06  ; #2腔体顶伸气缸下降位标志[0002.06]
ANDNOT 802.05  ; #2腔体顶伸气缸上升位标志[0002.05]
LD H32.05  ; 腔体有复测需求
ANDNOT H5.14  ; 测试模式（0-双检 1-单检）
AND H5.13  ; 复测模式（0-关闭 1-打开）
ORLD
ANDLD
LD 851.03  ; 进料伺服Z轴待机位标志
LD H24.00  ; 进料伺服X轴回原点记忆
ANDNOT 850.05  ; 进料伺服X轴#2腔放料位标志
LD 850.03  ; 进料伺服X轴取料位标志
OR 850.04  ; 进料伺服X轴#1腔放料位标志
OR 850.06  ; 进料伺服X轴#3腔放料位标志
OR 850.07  ; 进料伺服X轴#1夹爪扫码NG放料位标志
OR 850.08  ; 进料伺服X轴#2夹爪扫码NG放料位标志
OR 850.09  ; 进料伺服X轴#1夹爪配对取放料位标志
OR 850.10  ; 进料伺服X轴#2夹爪配对取放料位标志
ANDLD
ORLD
ANDLD
LD 853.03  ; 出料伺服Z轴待机位标志
LD H44.00  ; 出料伺服X轴回原点记忆
ANDNOT 852.05  ; 出料伺服X轴#2腔取料位标志
LD 852.03  ; 出料伺服X轴放料位标志
OR 852.04  ; 出料伺服X轴#1腔取料位标志
OR 852.06  ; 出料伺服X轴#3腔取料位标志
OR 852.07  ; 出料伺服X轴#1夹爪氦检NG放料位标志
OR 852.08  ; 出料伺服X轴#2夹爪氦检NG放料位标志
OR 852.09  ; 出料伺服X轴#1夹爪配对取放料位标志
OR 852.10  ; 出料伺服X轴#2夹爪配对取放料位标志
ANDLD
ORLD
ANDLD
OUT D1092.00  ; #2腔体机构平移气缸安全移动条件

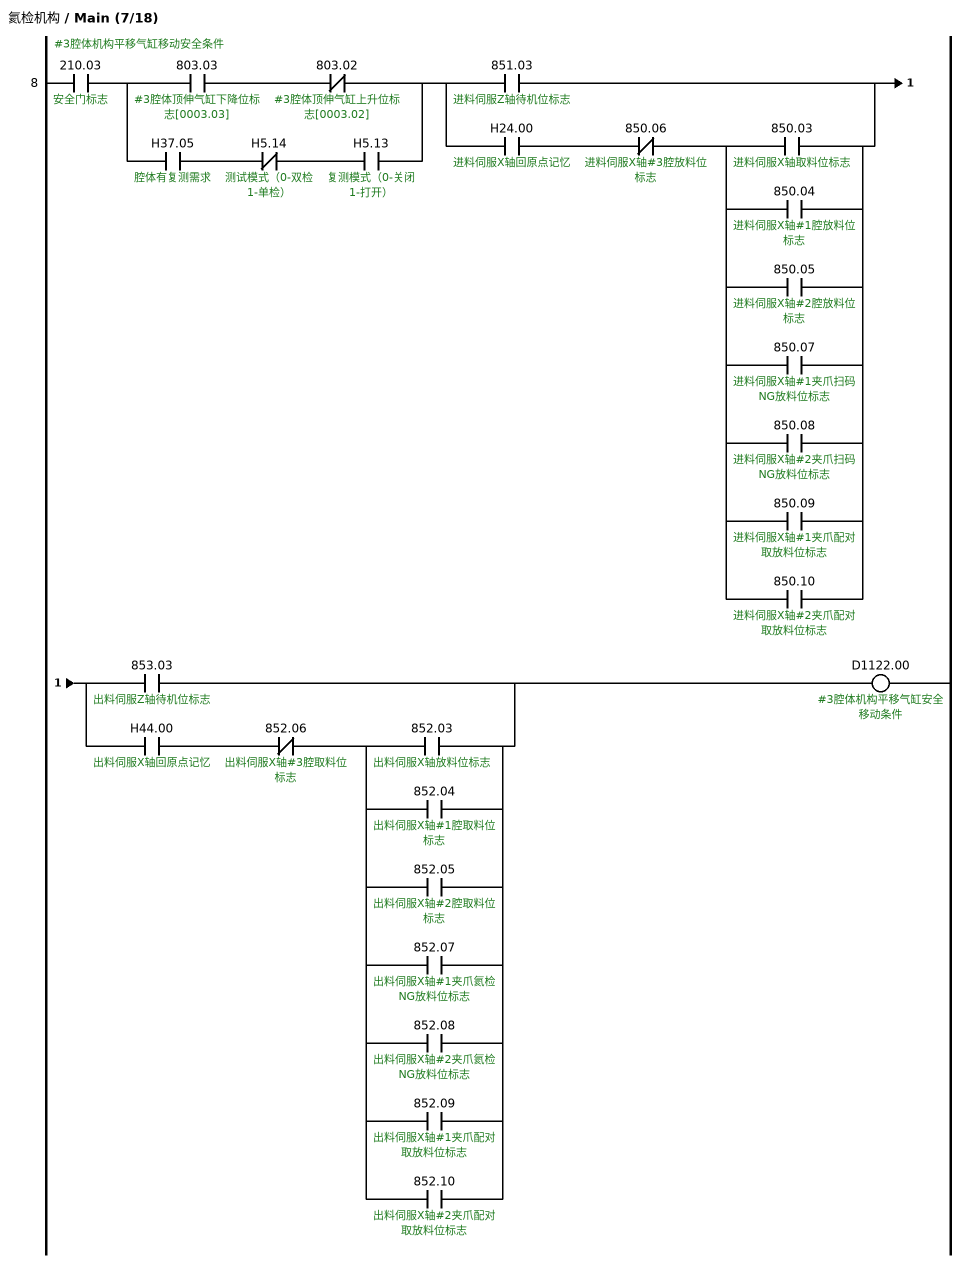
; rung 8: #3腔体机构平移气缸移动安全条件
LD 210.03  ; 安全门标志
LD 803.03  ; #3腔体顶伸气缸下降位标志[0003.03]
ANDNOT 803.02  ; #3腔体顶伸气缸上升位标志[0003.02]
LD H37.05  ; 腔体有复测需求
ANDNOT H5.14  ; 测试模式（0-双检 1-单检）
AND H5.13  ; 复测模式（0-关闭 1-打开）
ORLD
ANDLD
LD 851.03  ; 进料伺服Z轴待机位标志
LD H24.00  ; 进料伺服X轴回原点记忆
ANDNOT 850.06  ; 进料伺服X轴#3腔放料位标志
LD 850.03  ; 进料伺服X轴取料位标志
OR 850.04  ; 进料伺服X轴#1腔放料位标志
OR 850.05  ; 进料伺服X轴#2腔放料位标志
OR 850.07  ; 进料伺服X轴#1夹爪扫码NG放料位标志
OR 850.08  ; 进料伺服X轴#2夹爪扫码NG放料位标志
OR 850.09  ; 进料伺服X轴#1夹爪配对取放料位标志
OR 850.10  ; 进料伺服X轴#2夹爪配对取放料位标志
ANDLD
ORLD
ANDLD
LD 853.03  ; 出料伺服Z轴待机位标志
LD H44.00  ; 出料伺服X轴回原点记忆
ANDNOT 852.06  ; 出料伺服X轴#3腔取料位标志
LD 852.03  ; 出料伺服X轴放料位标志
OR 852.04  ; 出料伺服X轴#1腔取料位标志
OR 852.05  ; 出料伺服X轴#2腔取料位标志
OR 852.07  ; 出料伺服X轴#1夹爪氦检NG放料位标志
OR 852.08  ; 出料伺服X轴#2夹爪氦检NG放料位标志
OR 852.09  ; 出料伺服X轴#1夹爪配对取放料位标志
OR 852.10  ; 出料伺服X轴#2夹爪配对取放料位标志
ANDLD
ORLD
ANDLD
OUT D1122.00  ; #3腔体机构平移气缸安全移动条件

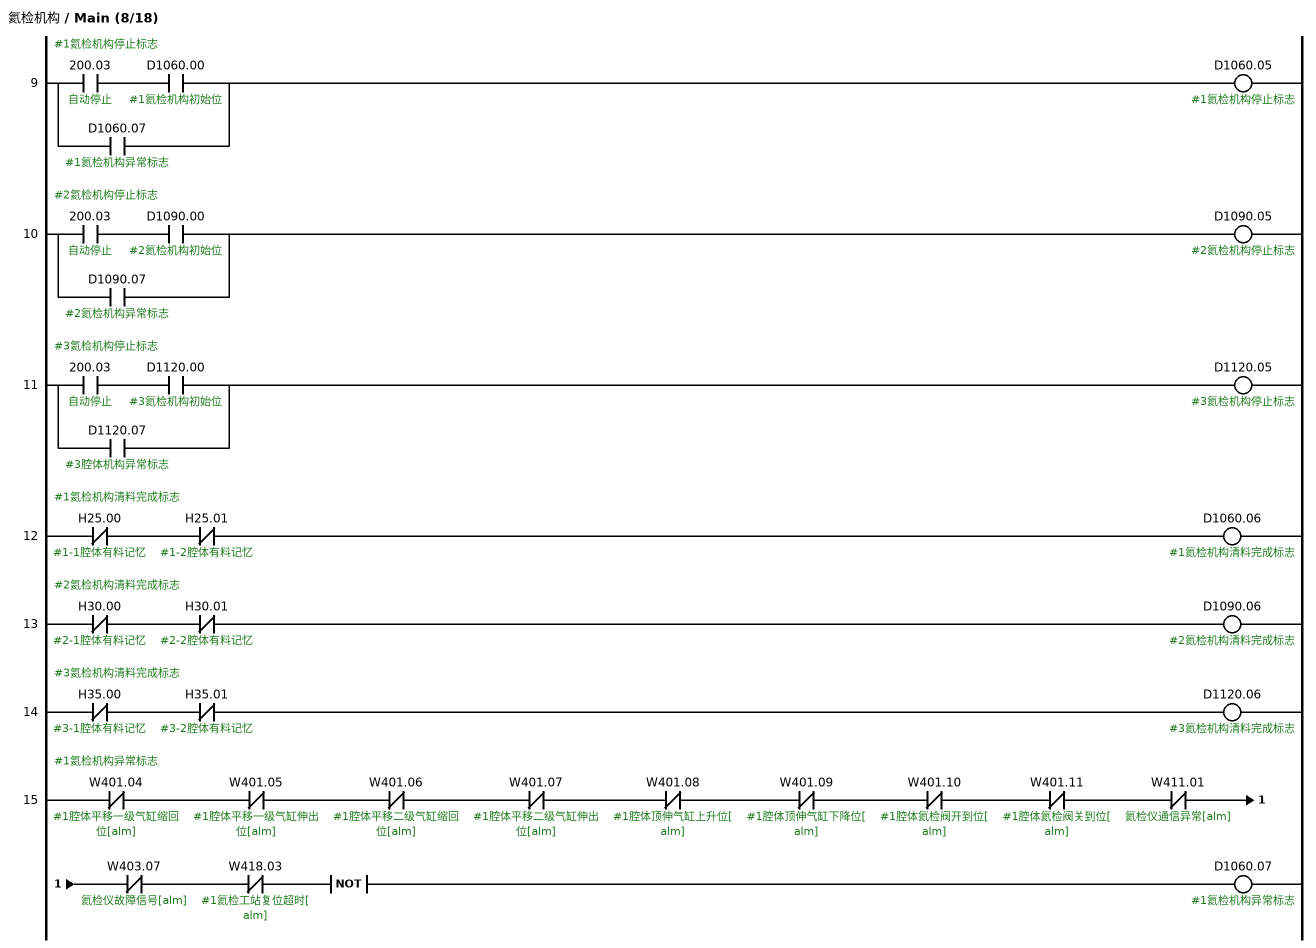
; rung 9: #1氦检机构停止标志
LD 200.03  ; 自动停止
AND D1060.00  ; #1氦检机构初始位
OR D1060.07  ; #1氦检机构异常标志
OUT D1060.05  ; #1氦检机构停止标志
; rung 10: #2氦检机构停止标志
LD 200.03  ; 自动停止
AND D1090.00  ; #2氦检机构初始位
OR D1090.07  ; #2氦检机构异常标志
OUT D1090.05  ; #2氦检机构停止标志
; rung 11: #3氦检机构停止标志
LD 200.03  ; 自动停止
AND D1120.00  ; #3氦检机构初始位
OR D1120.07  ; #3腔体机构异常标志
OUT D1120.05  ; #3氦检机构停止标志
; rung 12: #1氦检机构清料完成标志
LDNOT H25.00  ; #1-1腔体有料记忆
ANDNOT H25.01  ; #1-2腔体有料记忆
OUT D1060.06  ; #1氦检机构清料完成标志
; rung 13: #2氦检机构清料完成标志
LDNOT H30.00  ; #2-1腔体有料记忆
ANDNOT H30.01  ; #2-2腔体有料记忆
OUT D1090.06  ; #2氦检机构清料完成标志
; rung 14: #3氦检机构清料完成标志
LDNOT H35.00  ; #3-1腔体有料记忆
ANDNOT H35.01  ; #3-2腔体有料记忆
OUT D1120.06  ; #3氦检机构清料完成标志
; rung 15: #1氦检机构异常标志
LDNOT W401.04  ; #1腔体平移一级气缸缩回位[alm]
ANDNOT W401.05  ; #1腔体平移一级气缸伸出位[alm]
ANDNOT W401.06  ; #1腔体平移二级气缸缩回位[alm]
ANDNOT W401.07  ; #1腔体平移二级气缸伸出位[alm]
ANDNOT W401.08  ; #1腔体顶伸气缸上升位[alm]
ANDNOT W401.09  ; #1腔体顶伸气缸下降位[alm]
ANDNOT W401.10  ; #1腔体氦检阀开到位[alm]
ANDNOT W401.11  ; #1腔体氦检阀关到位[alm]
ANDNOT W411.01  ; 氦检仪通信异常[alm]
ANDNOT W403.07  ; 氦检仪故障信号[alm]
ANDNOT W418.03  ; #1氦检工站复位超时[alm]
NOT(520)
OUT D1060.07  ; #1氦检机构异常标志

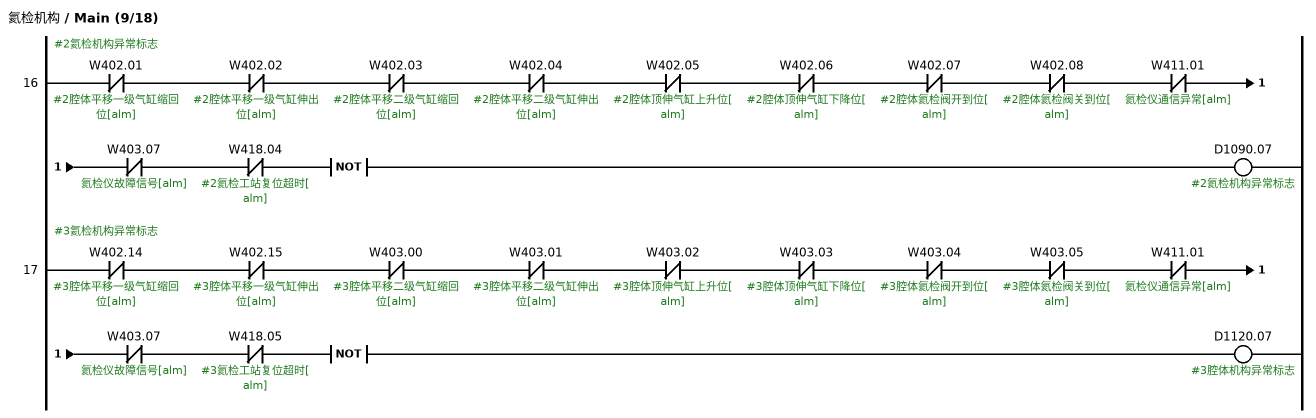
; rung 16: #2氦检机构异常标志
LDNOT W402.01  ; #2腔体平移一级气缸缩回位[alm]
ANDNOT W402.02  ; #2腔体平移一级气缸伸出位[alm]
ANDNOT W402.03  ; #2腔体平移二级气缸缩回位[alm]
ANDNOT W402.04  ; #2腔体平移二级气缸伸出位[alm]
ANDNOT W402.05  ; #2腔体顶伸气缸上升位[alm]
ANDNOT W402.06  ; #2腔体顶伸气缸下降位[alm]
ANDNOT W402.07  ; #2腔体氦检阀开到位[alm]
ANDNOT W402.08  ; #2腔体氦检阀关到位[alm]
ANDNOT W411.01  ; 氦检仪通信异常[alm]
ANDNOT W403.07  ; 氦检仪故障信号[alm]
ANDNOT W418.04  ; #2氦检工站复位超时[alm]
NOT(520)
OUT D1090.07  ; #2氦检机构异常标志
; rung 17: #3氦检机构异常标志
LDNOT W402.14  ; #3腔体平移一级气缸缩回位[alm]
ANDNOT W402.15  ; #3腔体平移一级气缸伸出位[alm]
ANDNOT W403.00  ; #3腔体平移二级气缸缩回位[alm]
ANDNOT W403.01  ; #3腔体平移二级气缸伸出位[alm]
ANDNOT W403.02  ; #3腔体顶伸气缸上升位[alm]
ANDNOT W403.03  ; #3腔体顶伸气缸下降位[alm]
ANDNOT W403.04  ; #3腔体氦检阀开到位[alm]
ANDNOT W403.05  ; #3腔体氦检阀关到位[alm]
ANDNOT W411.01  ; 氦检仪通信异常[alm]
ANDNOT W403.07  ; 氦检仪故障信号[alm]
ANDNOT W418.05  ; #3氦检工站复位超时[alm]
NOT(520)
OUT D1120.07  ; #3腔体机构异常标志

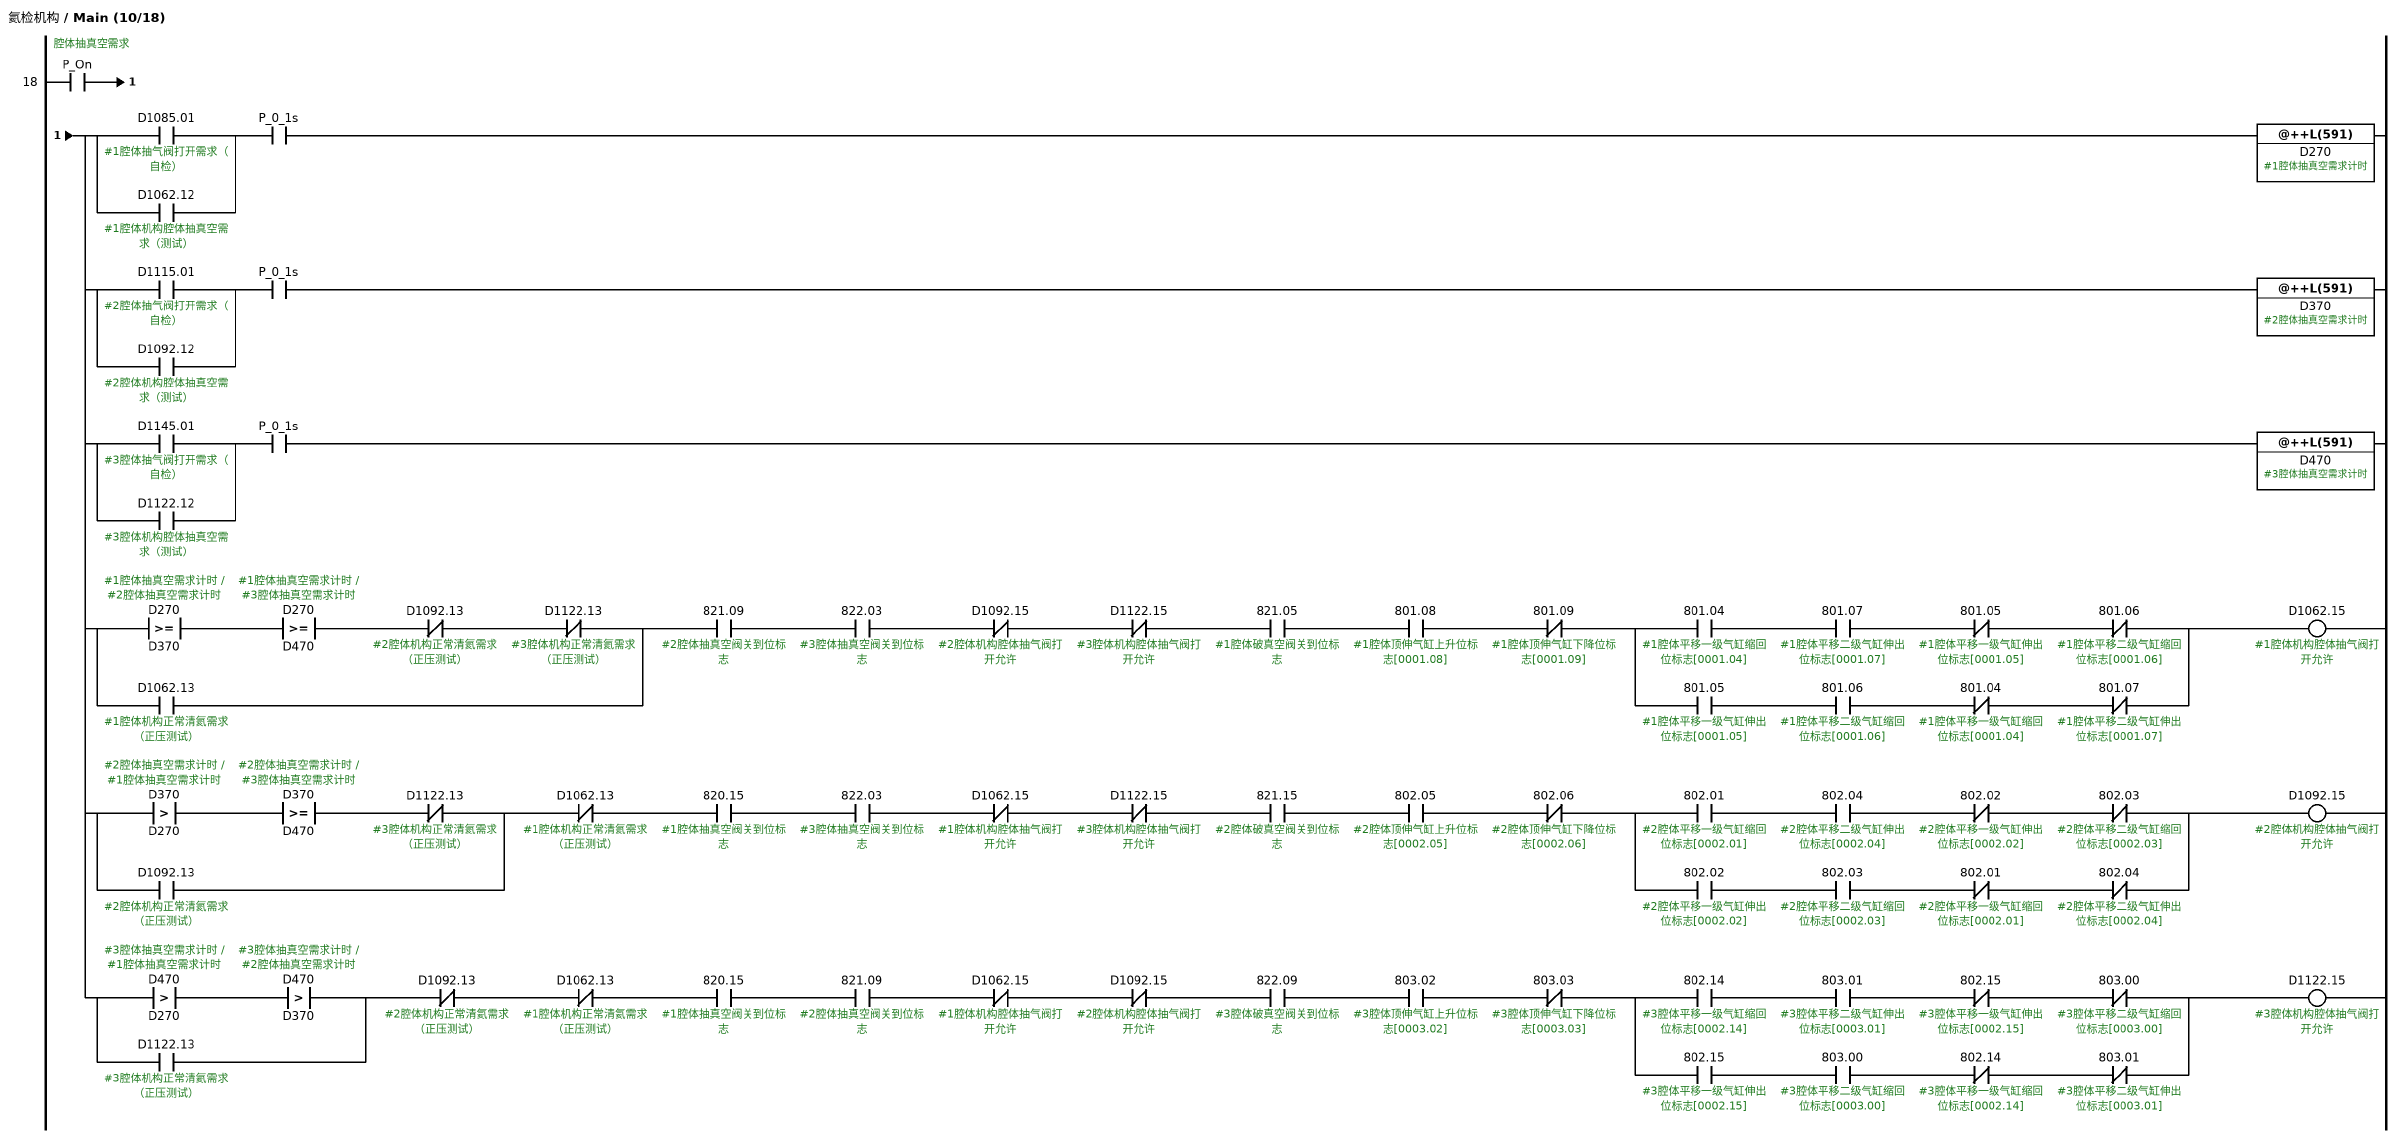
; rung 18: 腔体抽真空需求
LD P_On
OUT TR0
LD D1085.01  ; #1腔体抽气阀打开需求（自检）
OR D1062.12  ; #1腔体机构腔体抽真空需求（测试）
ANDLD
AND P_0_1s
@++L(591) D270  ; #1腔体抽真空需求计时
LD TR0
LD D1115.01  ; #2腔体抽气阀打开需求（自检）
OR D1092.12  ; #2腔体机构腔体抽真空需求（测试）
ANDLD
AND P_0_1s
@++L(591) D370  ; #2腔体抽真空需求计时
LD TR0
LD D1145.01  ; #3腔体抽气阀打开需求（自检）
OR D1122.12  ; #3腔体机构腔体抽真空需求（测试）
ANDLD
AND P_0_1s
@++L(591) D470  ; #3腔体抽真空需求计时
LD TR0
LD>=L(326) D270 D370  ; #1腔体抽真空需求计时, #2腔体抽真空需求计时
AND>=L(326) D270 D470  ; #1腔体抽真空需求计时, #3腔体抽真空需求计时
ANDNOT D1092.13  ; #2腔体机构正常清氦需求（正压测试）
ANDNOT D1122.13  ; #3腔体机构正常清氦需求（正压测试）
OR D1062.13  ; #1腔体机构正常清氦需求（正压测试）
ANDLD
AND 821.09  ; #2腔体抽真空阀关到位标志
AND 822.03  ; #3腔体抽真空阀关到位标志
ANDNOT D1092.15  ; #2腔体机构腔体抽气阀打开允许
ANDNOT D1122.15  ; #3腔体机构腔体抽气阀打开允许
AND 821.05  ; #1腔体破真空阀关到位标志
AND 801.08  ; #1腔体顶伸气缸上升位标志[0001.08]
ANDNOT 801.09  ; #1腔体顶伸气缸下降位标志[0001.09]
LD 801.04  ; #1腔体平移一级气缸缩回位标志[0001.04]
AND 801.07  ; #1腔体平移二级气缸伸出位标志[0001.07]
ANDNOT 801.05  ; #1腔体平移一级气缸伸出位标志[0001.05]
ANDNOT 801.06  ; #1腔体平移二级气缸缩回位标志[0001.06]
LD 801.05  ; #1腔体平移一级气缸伸出位标志[0001.05]
AND 801.06  ; #1腔体平移二级气缸缩回位标志[0001.06]
ANDNOT 801.04  ; #1腔体平移一级气缸缩回位标志[0001.04]
ANDNOT 801.07  ; #1腔体平移二级气缸伸出位标志[0001.07]
ORLD
ANDLD
OUT D1062.15  ; #1腔体机构腔体抽气阀打开允许
LD TR0
LD>L(321) D370 D270  ; #2腔体抽真空需求计时, #1腔体抽真空需求计时
AND>=L(326) D370 D470  ; #2腔体抽真空需求计时, #3腔体抽真空需求计时
ANDNOT D1122.13  ; #3腔体机构正常清氦需求（正压测试）
OR D1092.13  ; #2腔体机构正常清氦需求（正压测试）
ANDLD
ANDNOT D1062.13  ; #1腔体机构正常清氦需求（正压测试）
AND 820.15  ; #1腔体抽真空阀关到位标志
AND 822.03  ; #3腔体抽真空阀关到位标志
ANDNOT D1062.15  ; #1腔体机构腔体抽气阀打开允许
ANDNOT D1122.15  ; #3腔体机构腔体抽气阀打开允许
AND 821.15  ; #2腔体破真空阀关到位标志
AND 802.05  ; #2腔体顶伸气缸上升位标志[0002.05]
ANDNOT 802.06  ; #2腔体顶伸气缸下降位标志[0002.06]
LD 802.01  ; #2腔体平移一级气缸缩回位标志[0002.01]
AND 802.04  ; #2腔体平移二级气缸伸出位标志[0002.04]
ANDNOT 802.02  ; #2腔体平移一级气缸伸出位标志[0002.02]
ANDNOT 802.03  ; #2腔体平移二级气缸缩回位标志[0002.03]
LD 802.02  ; #2腔体平移一级气缸伸出位标志[0002.02]
AND 802.03  ; #2腔体平移二级气缸缩回位标志[0002.03]
ANDNOT 802.01  ; #2腔体平移一级气缸缩回位标志[0002.01]
ANDNOT 802.04  ; #2腔体平移二级气缸伸出位标志[0002.04]
ORLD
ANDLD
OUT D1092.15  ; #2腔体机构腔体抽气阀打开允许
LD TR0
LD>L(321) D470 D270  ; #3腔体抽真空需求计时, #1腔体抽真空需求计时
AND>L(321) D470 D370  ; #3腔体抽真空需求计时, #2腔体抽真空需求计时
OR D1122.13  ; #3腔体机构正常清氦需求（正压测试）
ANDLD
ANDNOT D1092.13  ; #2腔体机构正常清氦需求（正压测试）
ANDNOT D1062.13  ; #1腔体机构正常清氦需求（正压测试）
AND 820.15  ; #1腔体抽真空阀关到位标志
AND 821.09  ; #2腔体抽真空阀关到位标志
ANDNOT D1062.15  ; #1腔体机构腔体抽气阀打开允许
ANDNOT D1092.15  ; #2腔体机构腔体抽气阀打开允许
AND 822.09  ; #3腔体破真空阀关到位标志
AND 803.02  ; #3腔体顶伸气缸上升位标志[0003.02]
ANDNOT 803.03  ; #3腔体顶伸气缸下降位标志[0003.03]
LD 802.14  ; #3腔体平移一级气缸缩回位标志[0002.14]
AND 803.01  ; #3腔体平移二级气缸伸出位标志[0003.01]
ANDNOT 802.15  ; #3腔体平移一级气缸伸出位标志[0002.15]
ANDNOT 803.00  ; #3腔体平移二级气缸缩回位标志[0003.00]
LD 802.15  ; #3腔体平移一级气缸伸出位标志[0002.15]
AND 803.00  ; #3腔体平移二级气缸缩回位标志[0003.00]
ANDNOT 802.14  ; #3腔体平移一级气缸缩回位标志[0002.14]
ANDNOT 803.01  ; #3腔体平移二级气缸伸出位标志[0003.01]
ORLD
ANDLD
OUT D1122.15  ; #3腔体机构腔体抽气阀打开允许

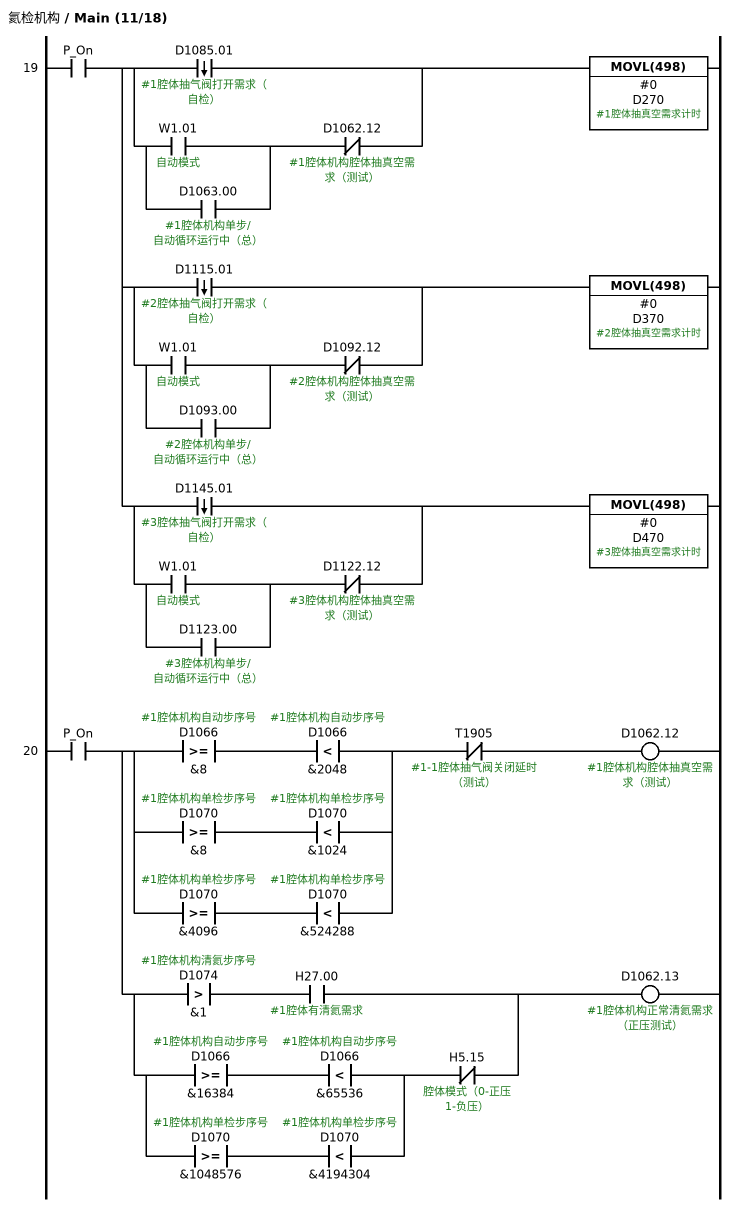
; rung 19
LD P_On
OUT TR0
%LD D1085.01  ; #1腔体抽气阀打开需求（自检）
LD W1.01  ; 自动模式
OR D1063.00  ; #1腔体机构单步/自动循环运行中（总）
ANDNOT D1062.12  ; #1腔体机构腔体抽真空需求（测试）
ORLD
ANDLD
MOVL(498) #0 D270  ; #1腔体抽真空需求计时
LD TR0
%LD D1115.01  ; #2腔体抽气阀打开需求（自检）
LD W1.01  ; 自动模式
OR D1093.00  ; #2腔体机构单步/自动循环运行中（总）
ANDNOT D1092.12  ; #2腔体机构腔体抽真空需求（测试）
ORLD
ANDLD
MOVL(498) #0 D370  ; #2腔体抽真空需求计时
LD TR0
%LD D1145.01  ; #3腔体抽气阀打开需求（自检）
LD W1.01  ; 自动模式
OR D1123.00  ; #3腔体机构单步/自动循环运行中（总）
ANDNOT D1122.12  ; #3腔体机构腔体抽真空需求（测试）
ORLD
ANDLD
MOVL(498) #0 D470  ; #3腔体抽真空需求计时
; rung 20
LD P_On
OUT TR0
LD>=L(326) D1066 &8  ; #1腔体机构自动步序号
AND<L(311) D1066 &2048  ; #1腔体机构自动步序号
LD>=L(326) D1070 &8  ; #1腔体机构单检步序号
AND<L(311) D1070 &1024  ; #1腔体机构单检步序号
ORLD
LD>=L(326) D1070 &4096  ; #1腔体机构单检步序号
AND<L(311) D1070 &524288  ; #1腔体机构单检步序号
ORLD
ANDLD
ANDNOT T1905  ; #1-1腔体抽气阀关闭延时（测试）
OUT D1062.12  ; #1腔体机构腔体抽真空需求（测试）
LD TR0
LD>L(321) D1074 &1  ; #1腔体机构清氦步序号
AND H27.00  ; #1腔体有清氦需求
LD>=L(326) D1066 &16384  ; #1腔体机构自动步序号
AND<L(311) D1066 &65536  ; #1腔体机构自动步序号
LD>=L(326) D1070 &1048576  ; #1腔体机构单检步序号
AND<L(311) D1070 &4194304  ; #1腔体机构单检步序号
ORLD
ANDNOT H5.15  ; 腔体模式（0-正压 1-负压）
ORLD
ANDLD
OUT D1062.13  ; #1腔体机构正常清氦需求（正压测试）

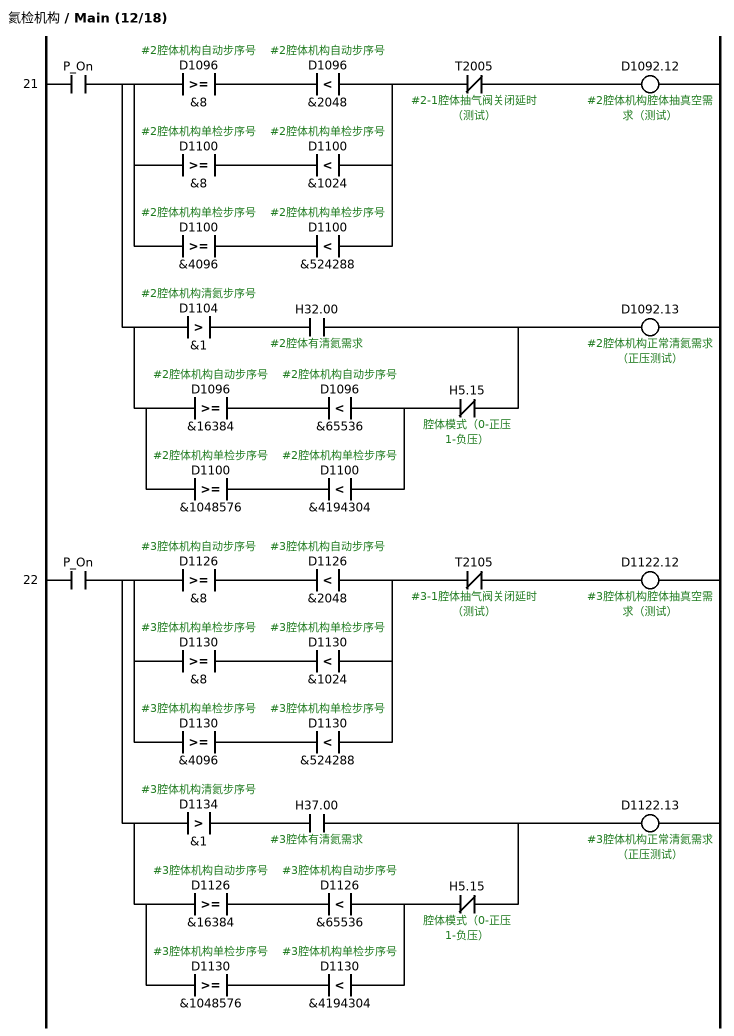
; rung 21
LD P_On
OUT TR0
LD>=L(326) D1096 &8  ; #2腔体机构自动步序号
AND<L(311) D1096 &2048  ; #2腔体机构自动步序号
LD>=L(326) D1100 &8  ; #2腔体机构单检步序号
AND<L(311) D1100 &1024  ; #2腔体机构单检步序号
ORLD
LD>=L(326) D1100 &4096  ; #2腔体机构单检步序号
AND<L(311) D1100 &524288  ; #2腔体机构单检步序号
ORLD
ANDLD
ANDNOT T2005  ; #2-1腔体抽气阀关闭延时（测试）
OUT D1092.12  ; #2腔体机构腔体抽真空需求（测试）
LD TR0
LD>L(321) D1104 &1  ; #2腔体机构清氦步序号
AND H32.00  ; #2腔体有清氦需求
LD>=L(326) D1096 &16384  ; #2腔体机构自动步序号
AND<L(311) D1096 &65536  ; #2腔体机构自动步序号
LD>=L(326) D1100 &1048576  ; #2腔体机构单检步序号
AND<L(311) D1100 &4194304  ; #2腔体机构单检步序号
ORLD
ANDNOT H5.15  ; 腔体模式（0-正压 1-负压）
ORLD
ANDLD
OUT D1092.13  ; #2腔体机构正常清氦需求（正压测试）
; rung 22
LD P_On
OUT TR0
LD>=L(326) D1126 &8  ; #3腔体机构自动步序号
AND<L(311) D1126 &2048  ; #3腔体机构自动步序号
LD>=L(326) D1130 &8  ; #3腔体机构单检步序号
AND<L(311) D1130 &1024  ; #3腔体机构单检步序号
ORLD
LD>=L(326) D1130 &4096  ; #3腔体机构单检步序号
AND<L(311) D1130 &524288  ; #3腔体机构单检步序号
ORLD
ANDLD
ANDNOT T2105  ; #3-1腔体抽气阀关闭延时（测试）
OUT D1122.12  ; #3腔体机构腔体抽真空需求（测试）
LD TR0
LD>L(321) D1134 &1  ; #3腔体机构清氦步序号
AND H37.00  ; #3腔体有清氦需求
LD>=L(326) D1126 &16384  ; #3腔体机构自动步序号
AND<L(311) D1126 &65536  ; #3腔体机构自动步序号
LD>=L(326) D1130 &1048576  ; #3腔体机构单检步序号
AND<L(311) D1130 &4194304  ; #3腔体机构单检步序号
ORLD
ANDNOT H5.15  ; 腔体模式（0-正压 1-负压）
ORLD
ANDLD
OUT D1122.13  ; #3腔体机构正常清氦需求（正压测试）

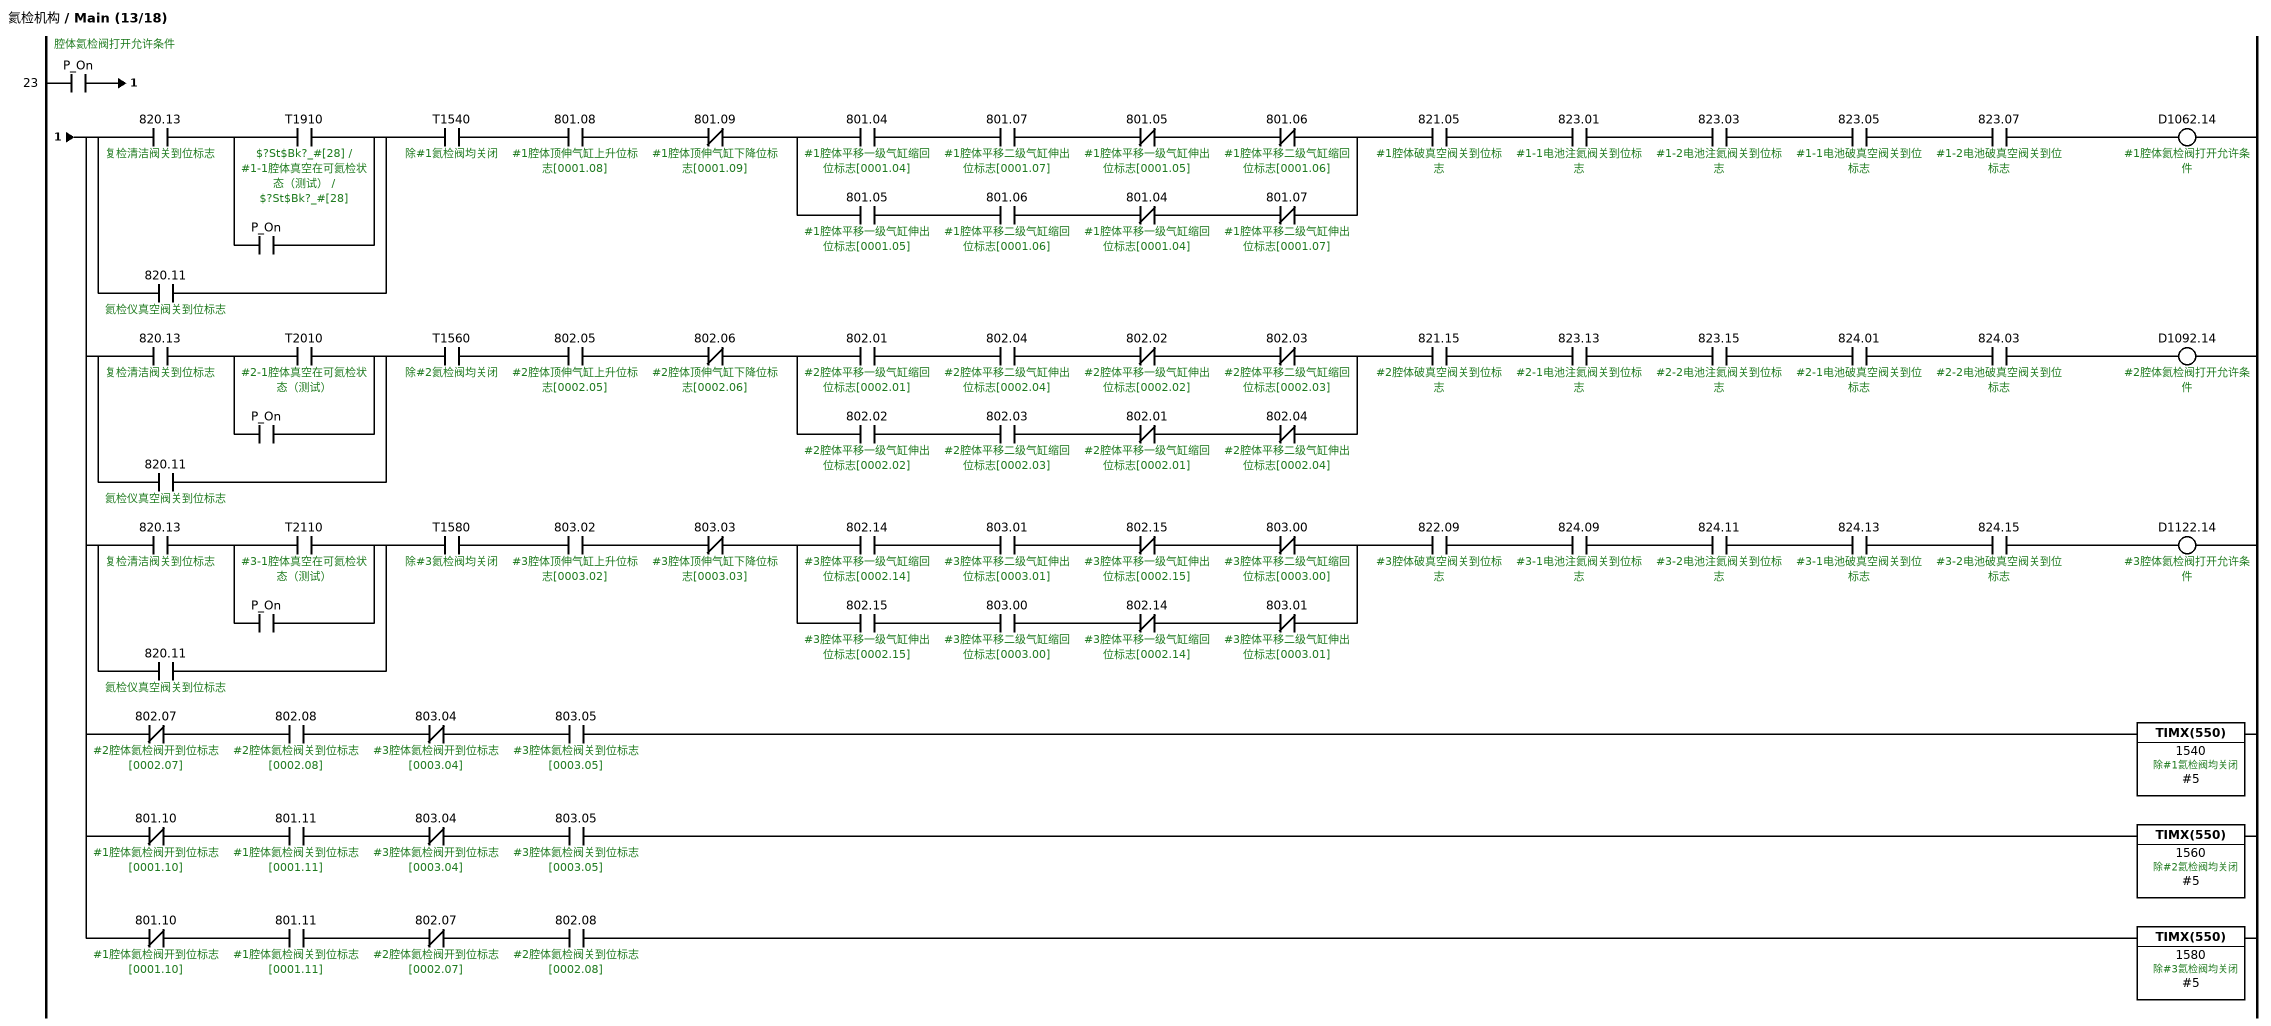
; rung 23: 腔体氦检阀打开允许条件
LD P_On
OUT TR0
LD 820.13  ; 复检清洁阀关到位标志
LD T1910  ; $?St$Bk?_#[28] / #1-1腔体真空在可氦检状态（测试） / $?St$Bk?_#[28]
OR P_On
ANDLD
OR 820.11  ; 氦检仪真空阀关到位标志
ANDLD
AND T1540  ; 除#1氦检阀均关闭
AND 801.08  ; #1腔体顶伸气缸上升位标志[0001.08]
ANDNOT 801.09  ; #1腔体顶伸气缸下降位标志[0001.09]
LD 801.04  ; #1腔体平移一级气缸缩回位标志[0001.04]
AND 801.07  ; #1腔体平移二级气缸伸出位标志[0001.07]
ANDNOT 801.05  ; #1腔体平移一级气缸伸出位标志[0001.05]
ANDNOT 801.06  ; #1腔体平移二级气缸缩回位标志[0001.06]
LD 801.05  ; #1腔体平移一级气缸伸出位标志[0001.05]
AND 801.06  ; #1腔体平移二级气缸缩回位标志[0001.06]
ANDNOT 801.04  ; #1腔体平移一级气缸缩回位标志[0001.04]
ANDNOT 801.07  ; #1腔体平移二级气缸伸出位标志[0001.07]
ORLD
ANDLD
AND 821.05  ; #1腔体破真空阀关到位标志
AND 823.01  ; #1-1电池注氦阀关到位标志
AND 823.03  ; #1-2电池注氦阀关到位标志
AND 823.05  ; #1-1电池破真空阀关到位标志
AND 823.07  ; #1-2电池破真空阀关到位标志
OUT D1062.14  ; #1腔体氦检阀打开允许条件
LD TR0
LD 820.13  ; 复检清洁阀关到位标志
LD T2010  ; #2-1腔体真空在可氦检状态（测试）
OR P_On
ANDLD
OR 820.11  ; 氦检仪真空阀关到位标志
ANDLD
AND T1560  ; 除#2氦检阀均关闭
AND 802.05  ; #2腔体顶伸气缸上升位标志[0002.05]
ANDNOT 802.06  ; #2腔体顶伸气缸下降位标志[0002.06]
LD 802.01  ; #2腔体平移一级气缸缩回位标志[0002.01]
AND 802.04  ; #2腔体平移二级气缸伸出位标志[0002.04]
ANDNOT 802.02  ; #2腔体平移一级气缸伸出位标志[0002.02]
ANDNOT 802.03  ; #2腔体平移二级气缸缩回位标志[0002.03]
LD 802.02  ; #2腔体平移一级气缸伸出位标志[0002.02]
AND 802.03  ; #2腔体平移二级气缸缩回位标志[0002.03]
ANDNOT 802.01  ; #2腔体平移一级气缸缩回位标志[0002.01]
ANDNOT 802.04  ; #2腔体平移二级气缸伸出位标志[0002.04]
ORLD
ANDLD
AND 821.15  ; #2腔体破真空阀关到位标志
AND 823.13  ; #2-1电池注氦阀关到位标志
AND 823.15  ; #2-2电池注氦阀关到位标志
AND 824.01  ; #2-1电池破真空阀关到位标志
AND 824.03  ; #2-2电池破真空阀关到位标志
OUT D1092.14  ; #2腔体氦检阀打开允许条件
LD TR0
LD 820.13  ; 复检清洁阀关到位标志
LD T2110  ; #3-1腔体真空在可氦检状态（测试）
OR P_On
ANDLD
OR 820.11  ; 氦检仪真空阀关到位标志
ANDLD
AND T1580  ; 除#3氦检阀均关闭
AND 803.02  ; #3腔体顶伸气缸上升位标志[0003.02]
ANDNOT 803.03  ; #3腔体顶伸气缸下降位标志[0003.03]
LD 802.14  ; #3腔体平移一级气缸缩回位标志[0002.14]
AND 803.01  ; #3腔体平移二级气缸伸出位标志[0003.01]
ANDNOT 802.15  ; #3腔体平移一级气缸伸出位标志[0002.15]
ANDNOT 803.00  ; #3腔体平移二级气缸缩回位标志[0003.00]
LD 802.15  ; #3腔体平移一级气缸伸出位标志[0002.15]
AND 803.00  ; #3腔体平移二级气缸缩回位标志[0003.00]
ANDNOT 802.14  ; #3腔体平移一级气缸缩回位标志[0002.14]
ANDNOT 803.01  ; #3腔体平移二级气缸伸出位标志[0003.01]
ORLD
ANDLD
AND 822.09  ; #3腔体破真空阀关到位标志
AND 824.09  ; #3-1电池注氦阀关到位标志
AND 824.11  ; #3-2电池注氦阀关到位标志
AND 824.13  ; #3-1电池破真空阀关到位标志
AND 824.15  ; #3-2电池破真空阀关到位标志
OUT D1122.14  ; #3腔体氦检阀打开允许条件
LD TR0
ANDNOT 802.07  ; #2腔体氦检阀开到位标志[0002.07]
AND 802.08  ; #2腔体氦检阀关到位标志[0002.08]
ANDNOT 803.04  ; #3腔体氦检阀开到位标志[0003.04]
AND 803.05  ; #3腔体氦检阀关到位标志[0003.05]
TIMX(550) 1540 #5  ; 除#1氦检阀均关闭
LD TR0
ANDNOT 801.10  ; #1腔体氦检阀开到位标志[0001.10]
AND 801.11  ; #1腔体氦检阀关到位标志[0001.11]
ANDNOT 803.04  ; #3腔体氦检阀开到位标志[0003.04]
AND 803.05  ; #3腔体氦检阀关到位标志[0003.05]
TIMX(550) 1560 #5  ; 除#2氦检阀均关闭
LD TR0
ANDNOT 801.10  ; #1腔体氦检阀开到位标志[0001.10]
AND 801.11  ; #1腔体氦检阀关到位标志[0001.11]
ANDNOT 802.07  ; #2腔体氦检阀开到位标志[0002.07]
AND 802.08  ; #2腔体氦检阀关到位标志[0002.08]
TIMX(550) 1580 #5  ; 除#3氦检阀均关闭

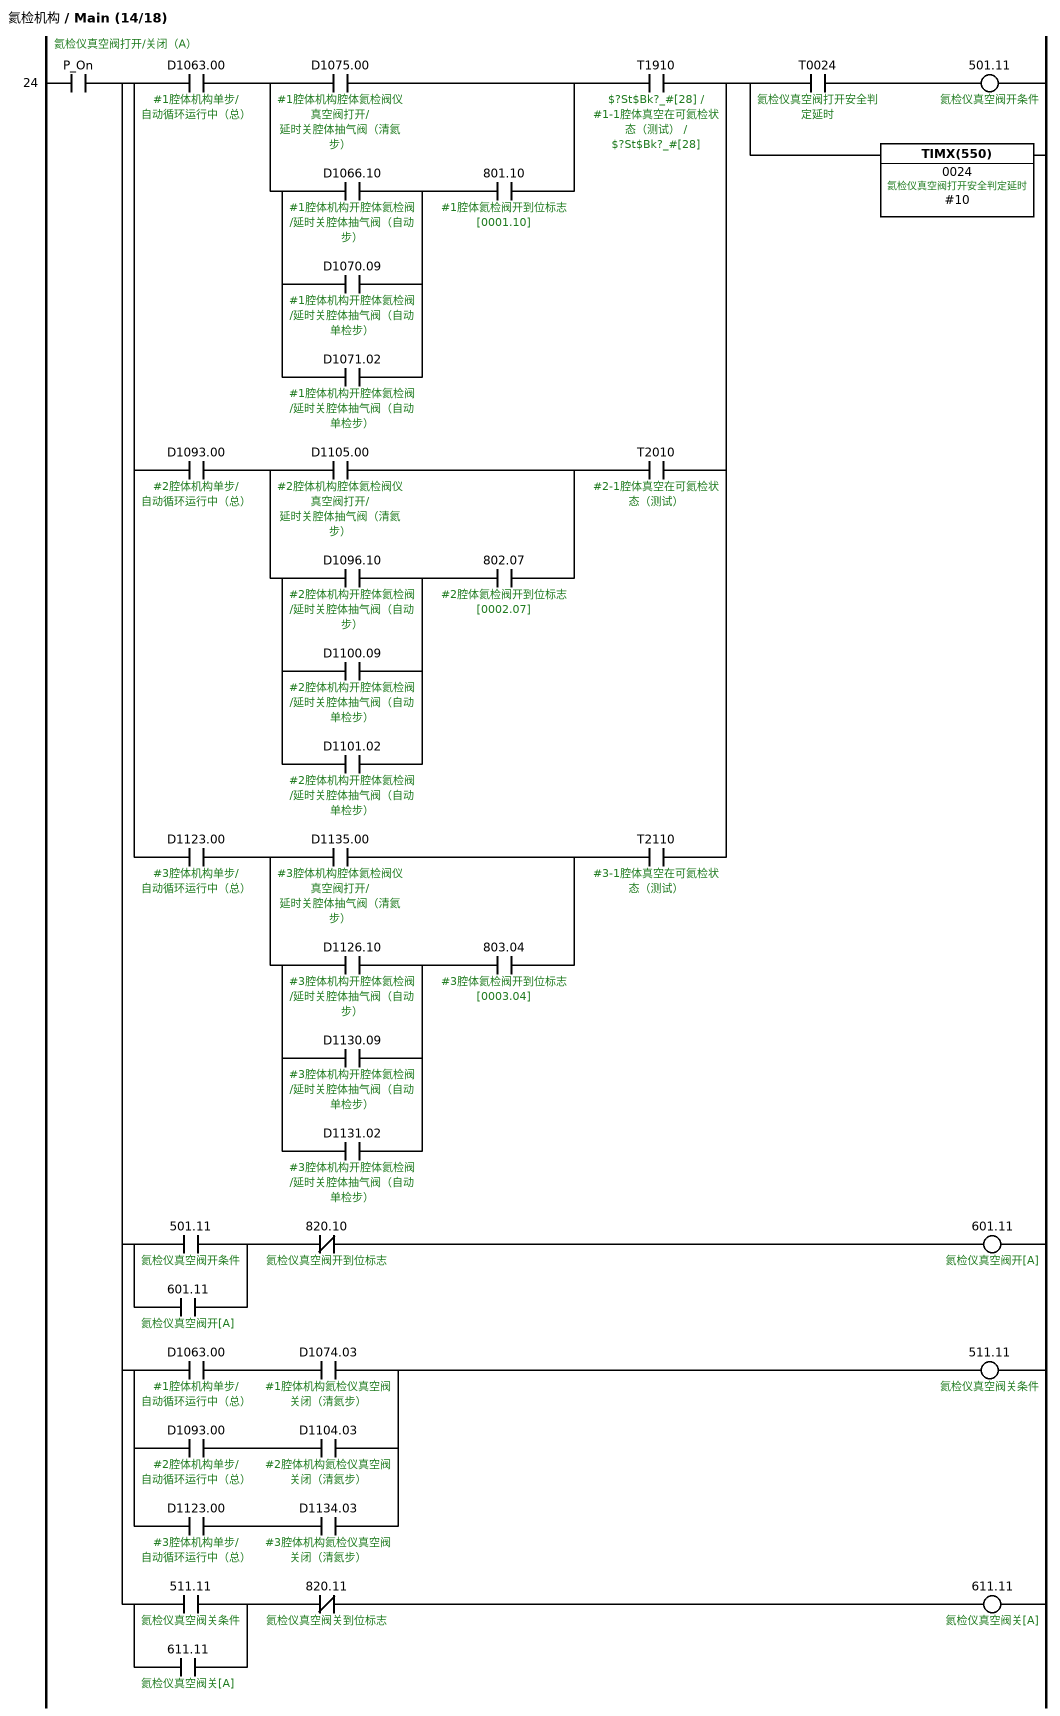
; rung 24: 氦检仪真空阀打开/关闭（A）
LD P_On
OUT TR0
LD D1063.00  ; #1腔体机构单步/自动循环运行中（总）
LD D1075.00  ; #1腔体机构腔体氦检阀仪真空阀打开/延时关腔体抽气阀（清氦步）
LD D1066.10  ; #1腔体机构开腔体氦检阀/延时关腔体抽气阀（自动步）
OR D1070.09  ; #1腔体机构开腔体氦检阀/延时关腔体抽气阀（自动单检步）
OR D1071.02  ; #1腔体机构开腔体氦检阀/延时关腔体抽气阀（自动单检步）
AND 801.10  ; #1腔体氦检阀开到位标志[0001.10]
ORLD
ANDLD
AND T1910  ; $?St$Bk?_#[28] / #1-1腔体真空在可氦检状态（测试） / $?St$Bk?_#[28]
LD D1093.00  ; #2腔体机构单步/自动循环运行中（总）
LD D1105.00  ; #2腔体机构腔体氦检阀仪真空阀打开/延时关腔体抽气阀（清氦步）
LD D1096.10  ; #2腔体机构开腔体氦检阀/延时关腔体抽气阀（自动步）
OR D1100.09  ; #2腔体机构开腔体氦检阀/延时关腔体抽气阀（自动单检步）
OR D1101.02  ; #2腔体机构开腔体氦检阀/延时关腔体抽气阀（自动单检步）
AND 802.07  ; #2腔体氦检阀开到位标志[0002.07]
ORLD
ANDLD
AND T2010  ; #2-1腔体真空在可氦检状态（测试）
ORLD
LD D1123.00  ; #3腔体机构单步/自动循环运行中（总）
LD D1135.00  ; #3腔体机构腔体氦检阀仪真空阀打开/延时关腔体抽气阀（清氦步）
LD D1126.10  ; #3腔体机构开腔体氦检阀/延时关腔体抽气阀（自动步）
OR D1130.09  ; #3腔体机构开腔体氦检阀/延时关腔体抽气阀（自动单检步）
OR D1131.02  ; #3腔体机构开腔体氦检阀/延时关腔体抽气阀（自动单检步）
AND 803.04  ; #3腔体氦检阀开到位标志[0003.04]
ORLD
ANDLD
AND T2110  ; #3-1腔体真空在可氦检状态（测试）
ORLD
ANDLD
OUT TR1
AND T0024  ; 氦检仪真空阀打开安全判定延时
OUT 501.11  ; 氦检仪真空阀开条件
LD TR1
TIMX(550) 0024 #10  ; 氦检仪真空阀打开安全判定延时
LD TR0
LD 501.11  ; 氦检仪真空阀开条件
OR 601.11  ; 氦检仪真空阀开[A]
ANDLD
ANDNOT 820.10  ; 氦检仪真空阀开到位标志
OUT 601.11  ; 氦检仪真空阀开[A]
LD TR0
LD D1063.00  ; #1腔体机构单步/自动循环运行中（总）
AND D1074.03  ; #1腔体机构氦检仪真空阀关闭（清氦步）
LD D1093.00  ; #2腔体机构单步/自动循环运行中（总）
AND D1104.03  ; #2腔体机构氦检仪真空阀关闭（清氦步）
ORLD
LD D1123.00  ; #3腔体机构单步/自动循环运行中（总）
AND D1134.03  ; #3腔体机构氦检仪真空阀关闭（清氦步）
ORLD
ANDLD
OUT 511.11  ; 氦检仪真空阀关条件
LD TR0
LD 511.11  ; 氦检仪真空阀关条件
OR 611.11  ; 氦检仪真空阀关[A]
ANDLD
ANDNOT 820.11  ; 氦检仪真空阀关到位标志
OUT 611.11  ; 氦检仪真空阀关[A]

